# B&R Automation Studio project BR_ZBM1 (part 2)

#### Shiftregister.st - Shiftregister
```iecst
(********************************************************************
 * COPYRIGHT --
 ********************************************************************
 * Program: Shiftregister
 * File: ShiftregisterCyclic.st
 * Author: jorkes
 * Created: July 08, 2014
 ********************************************************************
 * Implementation of program Shiftregister
 ********************************************************************)

PROGRAM _INIT
	SHFTREG.typCounters.usChainCounter := 0;
	SHFTREG.typCounters.uiChainCnt16x16 := 0;
	SHFTREG.typCounters.usStartUpCntr := 0;
	SHFTREG.typCounters.bStartChainCntr := FALSE;
	bStartCnt := TRUE;

	//Preset
	SHFTREG.typCounters.usChainCounter := 0;
END_PROGRAM

PROGRAM _CYCLIC
	//==============================================================
	//Software met 2 x puls/grijper
	//Encoderpuls 1
	//==============================================================
	bEncPuls1 := FALSE;

	IF EDGENEG(MCU.typChain.status.bSetSpeedReached) THEN
		idxCntr := 0;
		bEncActive1 := FALSE;
	END_IF

	IF MCU.typChain.status.bSetSpeedReached OR TRUE THEN
		//#1
		IF EDGEPOS(MCU.typIN.bEncPuls1) AND NOT bEncActive1 THEN
			tiStop1 := T#0ms;
			tiStart1 := clock_ms();
			//Wacht weer op een volgende trigger. -> #2
			bEncActive1 := TRUE;

			//IF SHFTREG.typCounters.bStartChainCntr THEN
				//ringcounter 0-74
				//SHFTREG.typCounters.usChainCounter := (SHFTREG.typCounters.usChainCounter + 1) MOD (SHFTREG.uiGripperCnt);
			//END_IF

			//Meten van de gemiddelde tijd tussen twee grijpers.
//			IF NOT(bSubCounter) THEN
//				tiStart3 := tiStart1;
//				bSubCounter := TRUE;
//			ELSE
//				tiStop3 := tiStart1;
//				tiDiff3[idx_Diff3] := tiStop3 - tiStart3;
//
//				idx_Diff3 := (idx_Diff3 + 1) MOD 10;
//
//				tiDiff3Total := T#0ms;
//
//				FOR idx := 0 TO 9 DO
//					tiDiff3Total := tiDiff3Total + tiDiff3[idx];
//				END_FOR
//
//				tiDiff3Total := tiDiff3Total / 10;
//
//				IF idxCntr > 9 THEN
//					tiMusecSub := tiDiff3Total / 16;
//				ELSE
//					idxCntr := idxCntr + 1;
//					tiMusecSub := SHFTREG.tiDistanceBetweenGrippers / 16;
//				END_IF
//
//				bSubCounter := FALSE;
//			END_IF
		END_IF

		//Sla actuele tijd op.
		tiActual1 := clock_ms();

		//#2
		IF bEncActive1 THEN
			tiCheck1[idx_Diff1] := tiActual1 - tiStart1;
			//Controleer of de tweede puls van dezelfde grijper is en niet van de volgende.
			IF NOT(tiCheck1[idx_Diff1] > T#300ms) THEN
				//Als de volgende trigger binnen de 300ms valt dan is het dezelfde grijper.
				//IF EDGEPOS(MCU.typIN.bEncPuls1) THEN
				//	bStartEnc := TRUE;
				//END_IF
				//Controleer de trigger op de afgaande flank en sla de tijd op.
//				IF EDGENEG(MCU.typIN.bEncPuls1) THEN
//					tiStop1 := clock_ms();
//					tiDiff1 := tiStop1 - tiStart1;
//					//Als de tijd tussen opgaande en de afgaande flank groter is dan (100ms) genereer een puls met dubbele tijd.
//					IF tiDiff1 > T#100ms THEN
//						//Dubbele puls tijd.
//						//tpPulsEnc1.PT := T#10ms;
//						//Activeer puls.
//						//tpPulsEnc1.IN := TRUE;
//						//Wacht weer op een volgende trigger. -> #1
//						bEncActive1 := FALSE;
//						//Start de chaincounter bij de lange puls! -> #1
//						SHFTREG.typCounters.bStartChainCntr := TRUE;
//						//SHFTREG.typCounters.usChainCounter := 0;
//					END_IF
				IF EDGEPOS(MCU.typIN.bEncPuls1) THEN
					tiStop1 := clock_ms();
					tiDiff1 := tiStop1 - tiStart1;
					//Als de tijd tussen de twee triggerpulsen groter is dan (100ms) genereer een puls van 5ms.
					IF tiDiff1 > T#50ms THEN
						bEncPuls1 := TRUE;
						//Wacht weer op een volgende trigger. -> #1
						bEncActive1 := FALSE;
					END_IF
					idx_Diff1 := (idx_Diff1 + 1) MOD 75;
				ELSIF (tiCheck1[idx_Diff1] >= (T#149ms - T#30ms)) AND (tiStop1 = T#0ms) THEN //(T#149ms - T#30ms)) THEN
					// generate puls
					bEncPuls1 := TRUE;
					//Wacht weer op een volgende trigger. -> #1
					bEncActive1 := FALSE;
					//Start de chaincounter bij de lange puls! -> #1
					SHFTREG.typCounters.bStartChainCntr := TRUE;
					SHFTREG.typCounters.usChainCounter := 0;
					idx_Diff1 := (idx_Diff1 + 1) MOD 75;
				END_IF
			ELSE
				//Wacht weer op een volgende trigger. -> #1
				bEncActive1 := FALSE;
			END_IF
		END_IF
	END_IF

	IF EDGEPOS(bEncPuls1) THEN

		IF NOT(bSubCounter) THEN
			tiStart3 := clock_ms();
			bSubCounter := TRUE;
		ELSE
			tiStop3 := clock_ms();
			tiDiff3[idx_Diff3] := tiStop3 - tiStart3;

			idx_Diff3 := (idx_Diff3 + 1) MOD 10;

			tiDiff3Total := T#0ms;

			FOR idx := 0 TO 9 DO
				tiDiff3Total := tiDiff3Total + tiDiff3[idx];
			END_FOR

			tiDiff3Total := tiDiff3Total / 10;

			IF idxCntr > 9 THEN
				tiMusecSub := tiDiff3Total / 16;
			ELSE
				idxCntr := idxCntr + 1;
				tiMusecSub := SHFTREG.tiDistanceBetweenGrippers / 16;
			END_IF

			bSubCounter := FALSE;
		END_IF

		SHFTREG.typCounters.usChainCounter := (SHFTREG.typCounters.usChainCounter + 1) MOD (SHFTREG.uiGripperCnt);
	END_IF
		//#3
	IF EDGEPOS(MCU.typIN.bEncPuls2) AND NOT bEncActive2 THEN
		tiStart2 := clock_ms();
		//Wacht weer op een volgende trigger. -> #4
		bEncActive2 := TRUE;
	END_IF

	//Sla actuele tijd op.
	tiActual2 := clock_ms();

	//#4
	IF bEncActive2 THEN
		tiCheck2 := tiActual2 - tiStart2;
		//Controleer of de tweede puls van dezelfde grijper is en niet van de volgende.
		IF NOT(tiCheck2 > T#300ms) THEN
			//Als de volgende trigger binnen de 300ms valt dan is het dezelfde grijper.
			//Controleer de trigger op de afgaande flank en sla de tijd op.
			IF EDGENEG(MCU.typIN.bEncPuls2) THEN
				tiStop2 := clock_ms();
				tiDiff2 := tiStop2 - tiStart2;
				//Als de tijd tussen opgaande en de afgaande flank groter is dan (150ms) genereer een puls met dubbele tijd.
				IF tiDiff2 > T#100ms THEN
					//Dubbele puls tijd.
					tpPulsEnc2.PT := T#200ms;
					//Activeer puls.
					tpPulsEnc2.IN := TRUE;
					//Wacht weer op een volgende trigger. -> #3
					bEncActive2 := FALSE;
				END_IF
			ELSIF EDGEPOS(MCU.typIN.bEncPuls2) THEN
				tiStop2 := clock_ms();
				tiDiff2 := tiStop2 - tiStart2;
				//Als de tijd tussen de twee triggerpulsen groter is dan (50ms) genereer een puls van 100ms.
				IF tiDiff2 > T#50ms THEN
					//Dubbele puls tijd.
					tpPulsEnc2.PT := T#100ms;
					//Activeer puls.
					tpPulsEnc2.IN := TRUE;
					//Wacht weer op een volgende trigger. -> #3
					bEncActive2 := FALSE;
				END_IF
		END_IF		ELSE
			//Wacht weer op een volgende trigger. -> #3
			bEncActive2 := FALSE;
		END_IF
	END_IF

	PulsGenerator_0(tInit := bEncPuls1, enable := bGblSimulation OR MCU.typChain.status.bSetSpeedReached, sysTim := systemTime, tiHigh := T#1ms, tiLow := tiMusecSub);

	IF bEncPuls1 THEN
		SHFTREG.typCounters.uiChainCnt16x16 := SHFTREG.typCounters.uiChainCnt16x16 AND 240;
	END_IF

	IF EDGENEG(PulsGenerator_0.bOutput) THEN
		SHFTREG.typCounters.uiChainCnt16x16 := (SHFTREG.typCounters.uiChainCnt16x16 + 1) MOD 256;
		IF (SHFTREG.typCounters.uiChainCnt16x16 = 0) THEN
			SHFTREG.typCounters.usChainOffset := SHFTREG.typCounters.usChainCounter;
		END_IF
	END_IF

	//4 x cam & light triggers
	//	CamTrig_0(CamPos := 5, reset := MCU.typIN.bEncPuls1, trigger := EDGENEG(PulsGenerator_0.bOutput), tiPuls := T#30ms, tiDelay := T#15ms); //tiDelay = zie excel berekening Beschrijving software.xlsx
	//	CamTrig_1(CamPos := 10, reset := MCU.typIN.bEncPuls1, trigger := EDGENEG(PulsGenerator_0.bOutput), tiPuls := T#30ms, tiDelay := T#7ms);
	//	CamTrig_2(CamPos := 12, reset := MCU.typIN.bEncPuls1, trigger := EDGENEG(PulsGenerator_0.bOutput), tiPuls := T#30ms, tiDelay := T#11ms);
	//	CamTrig_3(CamPos := 2, reset := MCU.typIN.bEncPuls1, trigger := EDGENEG(PulsGenerator_0.bOutput), tiPuls := T#30ms, tiDelay := T#26ms);
	CamTrig_0(CamPos := Settings.CamPosition1, reset := bEncPuls1, trigger := EDGENEG(PulsGenerator_0.bOutput), tiPuls := INT_TO_TIME(Settings.CamPulseLength), tiDelay := INT_TO_TIME(Settings.CamDelay1), tiExtraLight := INT_TO_TIME(Settings.FlitsBefore)); //tiDelay = zie excel berekening Beschrijving software.xlsx
	CamTrig_1(CamPos := Settings.CamPosition2, reset := bEncPuls1, trigger := EDGENEG(PulsGenerator_0.bOutput), tiPuls := INT_TO_TIME(Settings.CamPulseLength), tiDelay := INT_TO_TIME(Settings.CamDelay2), tiExtraLight := INT_TO_TIME(Settings.FlitsBefore));
	CamTrig_2(CamPos := Settings.CamPosition3, reset := bEncPuls1, trigger := EDGENEG(PulsGenerator_0.bOutput), tiPuls := INT_TO_TIME(Settings.CamPulseLength), tiDelay := INT_TO_TIME(Settings.CamDelay3), tiExtraLight := INT_TO_TIME(Settings.FlitsBefore));
	CamTrig_3(CamPos := Settings.CamPosition4, reset := bEncPuls1, trigger := EDGENEG(PulsGenerator_0.bOutput), tiPuls := INT_TO_TIME(Settings.CamPulseLength), tiDelay := INT_TO_TIME(Settings.CamDelay4), tiExtraLight := INT_TO_TIME(Settings.FlitsBefore));

	MCU.typOUT.bLightTrigger1 := CamTrig_0.outLight;
	MCU.typOUT.bCamTrigger1 := CamTrig_0.outCam;
	MCU.typOUT.bLightTrigger2 := CamTrig_1.outLight;
	MCU.typOUT.bCamTrigger2 := CamTrig_1.outCam;
	MCU.typOUT.bLightTrigger3 := CamTrig_2.outLight;
	MCU.typOUT.bCamTrigger3 := CamTrig_2.outCam;
	MCU.typOUT.bLightTrigger4 := CamTrig_3.outLight;
	MCU.typOUT.bCamTrigger4 := CamTrig_3.outCam;

	//===============================
	//Software met kettingplaatjes
	//===============================
	//bEncPuls1 := MCU.typIN.bEncPuls1

	//Afhandelen van encodertrigger 1
//	IF EDGEPOS(bEncPuls1) AND NOT bFall_1 THEN
//		tiMusecStart4 := clock_ms();
//		IF toggle THEN
//			toggle := FALSE;
//			tiMusecStop3 := clock_ms();
//			tiMusecDiff3 := tiMusecStop3 - tiMusecStart1;
//			tiMusecSub := tiMusecDiff3 / 16;
//		END_IF
//
//		//get number of elapsed microseconds in current tick
//		tiMusecStart1 := clock_ms();
//
//		//Wait for first gripper (double length sensor puls)
//		IF SHFTREG.typCounters.bStartChainCntr THEN
//			//ringcounter 0-75
//			SHFTREG.typCounters.usChainCounter := (SHFTREG.typCounters.usChainCounter + 1) MOD (SHFTREG.uiGripperCnt);
//		ELSE
//			//startup counter. Only for completing average sensor measuring
//			SHFTREG.typCounters.usStartUpCntr := (SHFTREG.typCounters.usStartUpCntr + 1) MOD 255;
//		END_IF
//
//		//Variable prevends that falling edge is triggered first
//		bFall_1 := TRUE;
//	END_IF
//
//	IF EDGENEG(bEncPuls1) AND bFall_1 THEN
//		toggle := TRUE;
//
//		//get number of elapsed microseconds in current tick
//		tiMusecStop1 := clock_ms();
//		tiMusecDiff1 := tiMusecStop1 - tiMusecStart1;
//
//		AverageSens_0(index := SHFTREG.typCounters.usChainCounter, tiMeasure := tiMusecDiff1);
//
//		//First counter that takes care of detecting first gripper
//		IF SHFTREG.typCounters.usStartUpCntr > 9 THEN
//			AverageSens_0(enable := TRUE);
//			//Check if there was a 1.5 times of length of average sensor puls
//			//IF tiMusecDiff1 > ( (AverageSens_0.tiAverage * 3)/2) THEN
//			IF tiMusecDiff1 > ( (tiMusecDiff2 * 3)/2) THEN
//				tiMusecBetweenEncStart := clock_ms();
//				SHFTREG.typCounters.bStartChainCntr := TRUE;
//				SHFTREG.typCounters.usChainCounter := 0;
//			END_IF
//		END_IF
//
//		bFall_1 := FALSE;
//	END_IF
//
//	//Afhandelen van encodertrigger 2
//	IF EDGEPOS(bEncPuls2) AND NOT bFall_2 THEN
//		tiMusecStart2 := clock_ms();
//		bFall_2 := TRUE;
//	END_IF
//
//	IF EDGENEG(bEncPuls2) AND bFall_2 THEN
//		tiMusecStop2 := clock_ms();
//		tiMusecDiff2 := tiMusecStop2 - tiMusecStart2;
//
//		AverageSens_1(index := SHFTREG.typCounters.usChainCounter, tiMeasure := tiMusecDiff2);
//
//		//First counter that takes care of detecting first gripper
//		IF SHFTREG.typCounters.usStartUpCntr > 9 THEN
//			AverageSens_1(enable := TRUE);
//			//Check if there was a 1.5 times of length of average sensor puls
//			IF tiMusecDiff2 > ( (AverageSens_1.tiAverage * 3)/2) THEN
//				//Check if first sensor detected first gripper already
//
//				IF SHFTREG.typCounters.bStartChainCntr THEN
//					tiMusecBetweenEncStop := clock_ms();
//					//calculate time between encoder sensor, by measuring first grippper
//					tiMusecBetweenEncDiff[usCntr] := tiMusecBetweenEncStop - tiMusecBetweenEncStart;
//					usCntr := (usCntr + 1) MOD 100;
//				END_IF
//			END_IF
//		END_IF
//		bFall_2 := FALSE;
//	END_IF

	IF MCU.typInterface.State <> RUN THEN
		// Blink
		IF NOT tpBlink.Q THEN
			MCU.typOUT.bGreenLight := MCU.typOUT.bRedLight;
			MCU.typOUT.bRedLight := NOT MCU.typOUT.bRedLight;
		END_IF
		tpBlink(IN:=(NOT tpBlink.Q), PT:=T#500ms);
	ELSE
		IF bEncPuls1 THEN
			MCU.typOUT.bRedLight := TRUE;
			tiLastPuls := clock_ms();
		END_IF
		MCU.typOUT.bGreenLight := clock_ms() - tiLastPuls < T#400ms;
	END_IF

	// Reject Unit
	//usGripperIndex := ( SHFTREG.typCounters.usChainCounter + RU.usChainPos) MOD  SHFTREG.uiGripperCnt;
	usGripperIndex := ( SHFTREG.typCounters.usChainCounter + SHFTREG.uiGripperCnt - RU.usChainPos) MOD  SHFTREG.uiGripperCnt;
	IF SHFTREG.typGripper[usGripperIndex].bRejectActive THEN
		//RU.bAddFlower.SET1 := TRUE;
		IF RU.typSettings.usTimingBU16 MOD 16 = SHFTREG.typCounters.uiChainCnt16x16 MOD 16 THEN
			RU.typOUT.bActivateGripper := SHFTREG.typGripper[usGripperIndex].bRejectOnOff;
			//fbResetGripper( ThisGripper := SHFTREG.typGripper[usGripperIndex]);
			SHFTREG.typGripper[usGripperIndex].bRejectActive := FALSE;
			SHFTREG.typGripper[usGripperIndex].bRejectOnOff := FALSE;
		END_IF
	END_IF

	// Now check if a gripper is positioned for the BU
	FOR i := 0 TO 9 DO

		//JORKES
		usGripperIndex := ( SHFTREG.typCounters.usChainCounter + SHFTREG.uiGripperCnt - BU[i].usChainPos) MOD  SHFTREG.uiGripperCnt;

		IF NOT BU[i].typInterface.bEmptyCmd THEN
			BU[i].typInterface.bEmptyCmd := SHFTREG.typGripper[usGripperIndex].siEmptyBU = i;
			SHFTREG.typGripper[usGripperIndex].siEmptyBU := -1;
			AsArLogWrite_EmptyCmd(enable := TRUE, ident := arlogBASE_USER_LOG_IDENT, logLevel := 1, errornr := 50003, mem := ADR(i), len := SIZEOF(i), asciiString :=  ADR('Empty command received'));
		END_IF

		IF NOT BU[i].bAddFlower THEN
			//JORKES
			//usGripperIndex := ( SHFTREG.typCounters.usChainCounter + SHFTREG.uiGripperCnt - BU[i].usChainPos) MOD  SHFTREG.uiGripperCnt;
			BU[i].GripperControl.IN := FALSE;

			//IF EDGEPOS(BU[i].typInterface.bEmptyCmd) THEN
			//	AsArLogWrite_EmptyCmd(enable := TRUE, ident := arlogBASE_USER_LOG_IDENT, logLevel := 1, errornr := 50002, mem := 0, len := 0, asciiString :=  ADR('Bosunit empty cmd set'));
			//END_IF

			IF i = SHFTREG.typGripper[usGripperIndex].usSetTarget THEN
				//SHFTREG.typGripper[usGripperIndex].
				BU[i].bAddFlower := TRUE;
				BU[i].typInterface.iReceivePos := SHFTREG.typGripper[usGripperIndex].uiCorrection;
				IF SHFTREG.typGripper[usGripperIndex].bFast THEN
					BU[i].typInterface.usServoSpeed := BU[i].typSettings.usFastSpeed;
				ELSE
					BU[i].typInterface.usServoSpeed := BU[i].typSettings.usSpeed;
				END_IF
				//////////BU[i].typSettings.usTimingBU16 := INT_TO_SINT( SHFTREG.typGripper[usGripperIndex].uiTimingBU16 MOD 16);
				// The gripper data is assigend
				//IF EDGEPOS(BU[i].bAddFlower) THEN
				//	AsArLogWrite_EmptyCmd(enable := TRUE, ident := arlogBASE_USER_LOG_IDENT, logLevel := 1, errornr := 50003, mem := ADR(i), len := SIZEOF(i), asciiString :=  ADR('Add flower'));
				//END_IF
			ELSE
				// The first gripper doen's contain a flow, does the
				usGripperIndex := ( SHFTREG.typCounters.usChainCounter - 1 + BU[i].usChainPos) MOD SHFTREG.uiGripperCnt;
				IF i = SHFTREG.typGripper[usGripperIndex].usSetTarget AND NOT BU[i].bBusyDrop THEN
					BU[i].typInterface.iReceivePos := SHFTREG.typGripper[usGripperIndex].uiCorrection;
				END_IF
			END_IF
		ELSE IF NOT BU[i].bBusyDrop THEN
			//JORKES
			//IF EDGEPOS(BU[i].rsActivateGripper.Q1) THEN
			IF EDGEPOS(BU[i].typSettings.usTimingBU16 = (SHFTREG.typCounters.uiChainCnt16x16 MOD 16) ) AND (i = SHFTREG.typGripper[usGripperIndex].usSetTarget) THEN
				fbResetGripper( ThisGripper := SHFTREG.typGripper[usGripperIndex]);
				BU[i].GripperControl.IN := TRUE;
				BU[i].bAddFlower := FALSE;
				END_IF
			END_IF

			//JORKES
			//BU[i].GripperControl.IN :=  BU[i].rsActivateGripper.Q1; // AND  i = SHFTREG.typGripper[usGripperIndex].usSetTarget;
			//BU[i].GripperControl.IN :=  BU[i].typSettings.usTimingBU16 = SHFTREG.typCounters.uiChainCnt16x16 MOD 16; // AND  i = SHFTREG.typGripper[usGripperIndex].usSetTarget;
		END_IF

		IF EDGENEG(BU[i].typOUT.bActivateGripper) THEN
		//	BU[i].bAddFlower(SET1 := FALSE, RESET := TRUE);
		END_IF
		//BU[i].GripperControl(tiSensDelay := BU[i].typInterface.tiDelayActiveGripper, tiSensPuls := INT_TO_TIME( Settings.BU_ActivateReleaseTime )); // T#3000ms); // Was 100 RSP
		BU[i].GripperControl( PT := INT_TO_TIME( Settings.BU_ActivateReleaseTime ));
		BU[i].typOUT.bActivateGripper := BU[i].GripperControl.Q OR  BU[i].typInterface.bManualGripperCmd;
		//JORKES
		//BU[i].rsActivateGripper(RESET1 := NOT BU[i].bAddFlower);
		//BU[i].GripperControl.IN :=  BU[i].rsActivateGripper.Q1;

		// TO DO
		// BU[i].bAddFlower.RESET := (i = SHFTREG.typGripper[usGripperIndex].usSetTarget);

	END_FOR
END_PROGRAM
```

#### Shiftregister.var - Local variables
```iecst
(********************************************************************
 * COPYRIGHT --
 ********************************************************************
 * Program: Shiftregister
 * File: Shiftregister.var
 * Author: jorkes
 * Created: July 08, 2014
 ********************************************************************
 * Local variables of program Shiftregister
 ********************************************************************)
(*Log*)
VAR
	AsArLogWrite_EmptyCmd : AsArLogWrite := (0);
	tiLastPuls : TIME;
END_VAR
(*Zonder kettingplaatjes*)
VAR
	bSubCounter : BOOL := FALSE;
	bEncPuls2 : BOOL;
	bEncPuls1 : BOOL;
	tpPulsEnc2 : TP;
	tpPulsEnc1 : TP;
	bEncActive1 : BOOL;
	bEncActive2 : BOOL;
	idxCntr : USINT := 0;
	idx : USINT := 0;
	idx_Diff1 : USINT := 0;
	idx_Diff3 : USINT := 0;
	tiActual2 : TIME;
	tiActual1 : TIME;
	tiCheck1 : ARRAY[0..74] OF TIME;
	tiDiff1 : TIME;
	tiStop1 : TIME;
	tiStart1 : TIME;
	tiCheck2 : TIME;
	tiDiff2 : TIME;
	tiStop2 : TIME;
	tiStart2 : TIME;
	tiCheck3 : TIME;
	tiDiff3Total : TIME;
	tiDiff3 : ARRAY[0..9] OF TIME;
	tiStop3 : TIME;
	tiStart3 : TIME;
END_VAR
(*Kettingteller*)
VAR
	bFall_1 : BOOL := FALSE;
	bFall_2 : BOOL := FALSE;
	tiMusecDiff2 : TIME;
	tiMusecDiff1 : TIME;
	tiMusecStart2 : TIME;
	tiMusecStart1 : TIME;
	tiMusecStop2 : TIME;
	tiMusecStop1 : TIME;
END_VAR
(*Kettingrek*)
VAR
	usCntr : USINT := 0;
	tiMusecBetweenEncDiff : ARRAY[0..100] OF TIME;
	tiMusecBetweenEncStop : TIME;
	tiMusecBetweenEncStart : TIME;
	AverageSens_1 : fbAverage;
	AverageSens_0 : fbAverage;
END_VAR
(*Grijper*)
VAR
	tiMusecSub : TIME := T#600ms;
	tiMusecDiff3 : TIME;
	tiMusecStop3 : TIME;
	toggle : BOOL;
END_VAR
(*Subcounter*)
VAR
	bStartCnt : BOOL;
	tiMusecDiff4 : TIME;
	tiMusecActual4 : TIME;
	PulsGenerator_0 : PulsGenerator;
	tiMusecStart4 : TIME;
	CamTrig_0 : fbTriggerBuf;
	CamTrig_1 : fbTriggerBuf;
	CamTrig_2 : fbTriggerBuf;
	CamTrig_3 : fbTriggerBuf;
END_VAR
(*Ligths*)
VAR
	tpBlink : TP;
END_VAR
(*BunchUnits*)
VAR
	i : USINT;
	usGripperIndex : USINT;
END_VAR
```

#### Shiftregister1.st - not listed in the package file held
```iecst
(********************************************************************
 * COPYRIGHT --
 ********************************************************************
 * Program: Shiftregister
 * File: ShiftregisterCyclic.st
 * Author: jorkes
 * Created: July 08, 2014
 ********************************************************************
 * Implementation of program Shiftregister
 ********************************************************************)

PROGRAM _INIT
	SHFTREG.typCounters.usChainCounter := 0;
	SHFTREG.typCounters.uiChainCnt16x16 := 0;
	SHFTREG.typCounters.usStartUpCntr := 0;
	SHFTREG.typCounters.bStartChainCntr := FALSE;
	bStartCnt := TRUE;
END_PROGRAM

PROGRAM _CYCLIC
	PulsGenerator_0(tInit := MCU.typIN.bEncPuls1, enable := bGblSimulation OR MCU.typInterface.State = RUN, sysTim := systemTime, tiHigh := T#1ms, tiLow := tiMusecSub);

	IF EDGENEG(PulsGenerator_0.bOutput) THEN
		SHFTREG.typCounters.uiChainCnt16x16 := (SHFTREG.typCounters.uiChainCnt16x16 + 1) MOD 256;
		IF (SHFTREG.typCounters.uiChainCnt16x16 = 0) THEN
			SHFTREG.typCounters.usChainOffset := SHFTREG.typCounters.usChainCounter;
		END_IF
	END_IF

	//4 x cam & light triggers
//	CamTrig_0(CamPos := 5, reset := MCU.typIN.bEncPuls1, trigger := EDGENEG(PulsGenerator_0.bOutput), tiPuls := T#30ms, tiDelay := T#15ms); //tiDelay = zie excel berekening Beschrijving software.xlsx
//	CamTrig_1(CamPos := 10, reset := MCU.typIN.bEncPuls1, trigger := EDGENEG(PulsGenerator_0.bOutput), tiPuls := T#30ms, tiDelay := T#7ms);
//	CamTrig_2(CamPos := 12, reset := MCU.typIN.bEncPuls1, trigger := EDGENEG(PulsGenerator_0.bOutput), tiPuls := T#30ms, tiDelay := T#11ms);
//	CamTrig_3(CamPos := 2, reset := MCU.typIN.bEncPuls1, trigger := EDGENEG(PulsGenerator_0.bOutput), tiPuls := T#30ms, tiDelay := T#26ms);
	CamTrig_0(CamPos := Settings.CamPosition1, reset := MCU.typIN.bEncPuls1, trigger := EDGENEG(PulsGenerator_0.bOutput), tiPuls := INT_TO_TIME(Settings.CamPulseLength), tiDelay := INT_TO_TIME(Settings.CamDelay1), tiExtraLight := INT_TO_TIME(Settings.FlitsBefore)); //tiDelay = zie excel berekening Beschrijving software.xlsx
	CamTrig_1(CamPos := Settings.CamPosition2, reset := MCU.typIN.bEncPuls1, trigger := EDGENEG(PulsGenerator_0.bOutput), tiPuls := INT_TO_TIME(Settings.CamPulseLength), tiDelay := INT_TO_TIME(Settings.CamDelay2), tiExtraLight := INT_TO_TIME(Settings.FlitsBefore));
	CamTrig_2(CamPos := Settings.CamPosition3, reset := MCU.typIN.bEncPuls1, trigger := EDGENEG(PulsGenerator_0.bOutput), tiPuls := INT_TO_TIME(Settings.CamPulseLength), tiDelay := INT_TO_TIME(Settings.CamDelay3), tiExtraLight := INT_TO_TIME(Settings.FlitsBefore));
	CamTrig_3(CamPos := Settings.CamPosition4, reset := MCU.typIN.bEncPuls1, trigger := EDGENEG(PulsGenerator_0.bOutput), tiPuls := INT_TO_TIME(Settings.CamPulseLength), tiDelay := INT_TO_TIME(Settings.CamDelay4), tiExtraLight := INT_TO_TIME(Settings.FlitsBefore));

	MCU.typOUT.bLightTrigger1 := CamTrig_0.outLight;
	MCU.typOUT.bCamTrigger1 := CamTrig_0.outCam;
	MCU.typOUT.bLightTrigger2 := CamTrig_1.outLight;
	MCU.typOUT.bCamTrigger2 := CamTrig_1.outCam;
	MCU.typOUT.bLightTrigger3 := CamTrig_2.outLight;
	MCU.typOUT.bCamTrigger3 := CamTrig_2.outCam;
	MCU.typOUT.bLightTrigger4 := CamTrig_3.outLight;
	MCU.typOUT.bCamTrigger4 := CamTrig_3.outCam;

	//Afhandelen van encodertrigger 1
	IF EDGEPOS(MCU.typIN.bEncPuls1) AND NOT bFall_1 THEN
		tiMusecStart4 := clock_ms();
		IF toggle THEN
			toggle := FALSE;
			tiMusecStop3 := clock_ms();
			tiMusecDiff3 := tiMusecStop3 - tiMusecStart1;
			tiMusecSub := tiMusecDiff3 / 16;
		END_IF

		//get number of elapsed microseconds in current tick
		tiMusecStart1 := clock_ms();

		//Wait for first gripper (double length sensor puls)
		IF SHFTREG.typCounters.bStartChainCntr THEN
			//ringcounter 0-75
			SHFTREG.typCounters.usChainCounter := (SHFTREG.typCounters.usChainCounter + 1) MOD (SHFTREG.uiGripperCnt);
		ELSE
			//startup counter. Only for completing average sensor measuring
			SHFTREG.typCounters.usStartUpCntr := (SHFTREG.typCounters.usStartUpCntr + 1) MOD 255;
		END_IF

		//Variable prevends that falling edge is triggered first
		bFall_1 := TRUE;
	END_IF

	IF EDGENEG(MCU.typIN.bEncPuls1) AND bFall_1 THEN
		toggle := TRUE;

		//get number of elapsed microseconds in current tick
		tiMusecStop1 := clock_ms();
		tiMusecDiff1 := tiMusecStop1 - tiMusecStart1;

		AverageSens_0(index := SHFTREG.typCounters.usChainCounter, tiMeasure := tiMusecDiff1);

		//First counter that takes care of detecting first gripper
		IF SHFTREG.typCounters.usStartUpCntr > 9 THEN
			AverageSens_0(enable := TRUE);
			//Check if there was a 1.5 times of length of average sensor puls
			IF tiMusecDiff1 > ( (AverageSens_0.tiAverage * 3)/2) THEN
				tiMusecBetweenEncStart := clock_ms();
				SHFTREG.typCounters.bStartChainCntr := TRUE;
			END_IF
		END_IF

		bFall_1 := FALSE;
	END_IF

	//Afhandelen van encodertrigger 2
	IF EDGEPOS(MCU.typIN.bEncPuls2) AND NOT bFall_2 THEN
		tiMusecStart2 := clock_ms();
		bFall_2 := TRUE;
	END_IF

	IF EDGENEG(MCU.typIN.bEncPuls2) AND bFall_2 THEN
		tiMusecStop2 := clock_ms();
		tiMusecDiff2 := tiMusecStop2 - tiMusecStart2;

		AverageSens_1(index := SHFTREG.typCounters.usChainCounter, tiMeasure := tiMusecDiff2);

		//First counter that takes care of detecting first gripper
		IF SHFTREG.typCounters.usStartUpCntr > 9 THEN
			AverageSens_1(enable := TRUE);
			//Check if there was a 1.5 times of length of average sensor puls
			IF tiMusecDiff2 > ( (AverageSens_1.tiAverage * 3)/2) THEN
				//Check if first sensor detected first gripper already
				IF SHFTREG.typCounters.bStartChainCntr THEN
					tiMusecBetweenEncStop := clock_ms();
					//calculate time between encoder sensor, by measuring first grippper
					tiMusecBetweenEncDiff[usCntr] := tiMusecBetweenEncStop - tiMusecBetweenEncStart;
					usCntr := (usCntr + 1) MOD 100;
				END_IF
			END_IF
		END_IF
		bFall_2 := FALSE;
	END_IF

	IF MCU.typInterface.State <> RUN THEN
		// Blink
		IF NOT tpBlink.Q THEN
			MCU.typOUT.bGreenLight := MCU.typOUT.bRedLight;
			MCU.typOUT.bRedLight := NOT MCU.typOUT.bRedLight;
		END_IF
		tpBlink(IN:=(NOT tpBlink.Q), PT:=T#500ms);
	ELSE
		MCU.typOUT.bRedLight := (MCU.typIN.bEncPuls1);
		MCU.typOUT.bGreenLight := TRUE;
	END_IF

	// Reject Unit
	//usGripperIndex := ( SHFTREG.typCounters.usChainCounter + RU.usChainPos) MOD  SHFTREG.uiGripperCnt;
	usGripperIndex := ( SHFTREG.typCounters.usChainCounter + SHFTREG.uiGripperCnt - RU.usChainPos) MOD  SHFTREG.uiGripperCnt;
	IF SHFTREG.typGripper[usGripperIndex].bRejectActive THEN
		//RU.srAddFlower.SET1 := TRUE;
		IF RU.typSettings.usTimingBU16 MOD 16 = SHFTREG.typCounters.uiChainCnt16x16 MOD 16 THEN
			RU.typOUT.bActivateGripper := SHFTREG.typGripper[usGripperIndex].bRejectOnOff;
			//fbResetGripper( ThisGripper := SHFTREG.typGripper[usGripperIndex]);
			SHFTREG.typGripper[usGripperIndex].bRejectActive := FALSE;
			SHFTREG.typGripper[usGripperIndex].bRejectOnOff := FALSE;
		END_IF
	END_IF

	// Now check if a gripper is positioned for the BU
	FOR i := 0 TO 1 DO

		usGripperIndex := ( SHFTREG.typCounters.usChainCounter + SHFTREG.uiGripperCnt - BU[i].usChainPos) MOD  SHFTREG.uiGripperCnt;
		//IF BU[i].typSettings.usTimingBU16 = SHFTREG.typCounters.uiChainCnt16x16 MOD 16 AND  i = SHFTREG.typGripper[usGripperIndex].usSetTarget THEN
		// The time has come to activate the grippers!!!
		//	BU[i].GripperControl.IN := TRUE;
		//END_IF

		IF NOT BU[i].srAddFlower THEN
			usGripperIndex := ( SHFTREG.typCounters.usChainCounter + SHFTREG.uiGripperCnt - BU[i].usChainPos) MOD  SHFTREG.uiGripperCnt;
		//	IF i = SHFTREG.typGripper[usGripperIndex].usSetTarget THEN
		//		// The first gripper doen's contain a flow, does the
		//		usGripperIndex := ( SHFTREG.typCounters.usChainCounter - 1 + BU[i].usChainPos) MOD  SHFTREG.uiGripperCnt;
		//		BU[i].typInterface.iReceivePos := SHFTREG.typGripper[usGripperIndex].uiCorrection;
		//	END_IF

			IF i = SHFTREG.typGripper[usGripperIndex].usSetTarget THEN
				//SHFTREG.typGripper[usGripperIndex].
				BU[i].srAddFlower := TRUE;
				BU[i].typInterface.bEmptyCmd := SHFTREG.typGripper[usGripperIndex].bEmptyBU;
				BU[i].typInterface.iReceivePos := SHFTREG.typGripper[usGripperIndex].uiCorrection;
				IF SHFTREG.typGripper[usGripperIndex].bFast THEN
					BU[i].typInterface.usServoSpeed := BU[i].typSettings.usFastSpeed;
				ELSE
					BU[i].typInterface.usServoSpeed := BU[i].typSettings.usSpeed;
				END_IF
				//////////BU[i].typSettings.usTimingBU16 := INT_TO_SINT( SHFTREG.typGripper[usGripperIndex].uiTimingBU16 MOD 16);
				// The gripper data is assigend

			END_IF
		ELSE
			// BU[i].srAddFlower.Q1 = TRUE so a flower is already assigned
			usGripperIndex := ( SHFTREG.typCounters.usChainCounter + SHFTREG.uiGripperCnt - BU[i].usChainPos) MOD  SHFTREG.uiGripperCnt;
			BU[i].rsActivateGripper.SET := BU[i].typSettings.usTimingBU16 = SHFTREG.typCounters.uiChainCnt16x16 MOD 16  AND  i = SHFTREG.typGripper[usGripperIndex].usSetTarget;

			//IF BU[i].typSettings.usTimingBU16 = SHFTREG.typCounters.uiChainCnt16x16 MOD 16 AND  i = SHFTREG.typGripper[usGripperIndex].usSetTarget THEN
				// The time has come to activate the grippers!!!
			//	BU[i].GripperControl.IN := TRUE;
			//END_IF
			IF EDGEPOS(BU[i].rsActivateGripper.Q1) THEN
				fbResetGripper( ThisGripper := SHFTREG.typGripper[usGripperIndex]);
			END_IF
			BU[i].GripperControl.IN :=  BU[i].rsActivateGripper.Q1; // AND  i = SHFTREG.typGripper[usGripperIndex].usSetTarget;
			//BU[i].GripperControl.IN :=  BU[i].typSettings.usTimingBU16 = SHFTREG.typCounters.uiChainCnt16x16 MOD 16; // AND  i = SHFTREG.typGripper[usGripperIndex].usSetTarget;
		END_IF

		IF EDGENEG(BU[i].typOUT.bActivateGripper) THEN
		//	BU[i].srAddFlower(SET1 := FALSE, RESET := TRUE);
		END_IF
		//BU[i].GripperControl(tiSensDelay := BU[i].typInterface.tiDelayActiveGripper, tiSensPuls := INT_TO_TIME( Settings.BU_ActivateReleaseTime )); // T#3000ms); // Was 100 RSP
		BU[i].GripperControl( PT := INT_TO_TIME( Settings.BU_ActivateReleaseTime ));
		BU[i].typOUT.bActivateGripper := BU[i].GripperControl.Q;
		BU[i].rsActivateGripper(RESET1 := NOT BU[i].srAddFlower);
		BU[i].GripperControl.IN :=  BU[i].rsActivateGripper.Q1;;
		// TO DO
		// 							BU[i].srAddFlower.RESET := (i = SHFTREG.typGripper[usGripperIndex].usSetTarget);

	END_FOR
END_PROGRAM
```

### Program Logical/MainControlUnit/Simulation (IEC) - Program

#### Simulation.st - Implementation code
```iecst
(********************************************************************
 * COPYRIGHT --
 ********************************************************************
 * Program: Simulation
 * File: Simulation.st
 * Author: jorkes
 * Created: July 08, 2014
 ********************************************************************
 * Implementation of program Init
 ********************************************************************)

PROGRAM _INIT
	typEncPuls1.tiHigh := tiEncPulsShort;
	typEncPuls1.tiLow := SHFTREG.tiDistanceBetweenGrippers - tiEncPulsShort;

	typEncPuls2.tiHigh := tiEncPulsShort;
	typEncPuls2.tiLow := SHFTREG.tiDistanceBetweenGrippers - tiEncPulsShort;
END_PROGRAM

PROGRAM _CYCLIC
	typEncPuls1(enable := bGblSimulation, sysTim := systemTime);
	typEncPuls2(enable := bGblSimulation, sysTim := systemTime);

	// In simulation the pulses are generated by the above function.
	IF bGblSimulation THEN
		MCU.typIN.bEncPuls1 := typEncPuls1.bOutput;
		MCU.typIN.bEncPuls2 := typEncPuls2.bOutput;
	END_IF

	IF SHFTREG.typCounters.bStartChainCntr THEN
		IF  SHFTREG.typCounters.usChainCounter >= (SHFTREG.uiGripperCnt - 1) THEN
			typEncPuls1.tiHigh := tiEncPulsLong;
			typEncPuls1.tiLow := SHFTREG.tiDistanceBetweenGrippers - tiEncPulsLong;
		ELSE
			typEncPuls1.tiHigh := tiEncPulsShort;
			typEncPuls1.tiLow := SHFTREG.tiDistanceBetweenGrippers - tiEncPulsShort;
		END_IF
	ELSE
		IF  SHFTREG.typCounters.usStartUpCntr >= 10 THEN
			typEncPuls1.tiHigh := tiEncPulsLong;
			typEncPuls1.tiLow := SHFTREG.tiDistanceBetweenGrippers - tiEncPulsLong;
		ELSE
			typEncPuls1.tiHigh := tiEncPulsShort;
			typEncPuls1.tiLow := SHFTREG.tiDistanceBetweenGrippers - tiEncPulsShort;
		END_IF
	END_IF

	IF SHFTREG.typCounters.usChainCounter = SHFTREG.typEncoder.uiEncSensorPosition2 THEN //Aantal grijpers tussen eerste en tweede encoder.
		typEncPuls2.tiHigh := tiEncPulsLong;
		typEncPuls2.tiLow := SHFTREG.tiDistanceBetweenGrippers - tiEncPulsLong;
	ELSE
		typEncPuls2.tiHigh := tiEncPulsShort;
		typEncPuls2.tiLow := SHFTREG.tiDistanceBetweenGrippers - tiEncPulsShort;
	END_IF

	//4 x cam & light triggers
	//Sensor_0(trigger := MCU.typIN.bEncPuls1, tiPuls := tiPulsCam, tiDelay := tiDelayCam_0);
	//Sensor_1(trigger := MCU.typIN.bEncPuls1, tiPuls := tiPulsCam, tiDelay := tiDelayCam_1);
	//Sensor_2(trigger := MCU.typIN.bEncPuls1, tiPuls := tiPulsCam, tiDelay := tiDelayCam_2);
	//Sensor_3(trigger := MCU.typIN.bEncPuls1, tiPuls := tiPulsCam, tiDelay := tiDelayCam_3);

	//MCU.typOUT.bCamTrigger1 := Sensor_0.outCam;
	//MCU.typOUT.bCamTrigger2 := Sensor_1.outCam;
	//MCU.typOUT.bCamTrigger3 := Sensor_2.outCam;
	//MCU.typOUT.bCamTrigger4 := Sensor_3.outCam;

	//MCU.typOUT.bLightTrigger1 := Sensor_0.outLight;
	//MCU.typOUT.bLightTrigger2 := Sensor_1.outLight;
	//MCU.typOUT.bLightTrigger3 := Sensor_2.outLight;
	//MCU.typOUT.bLightTrigger4 := Sensor_3.outLight;
END_PROGRAM
```

#### Simulation.var - Local variables
```iecst
(********************************************************************
 * COPYRIGHT --
 ********************************************************************
 * Program: Init
 * File: Init.var
 * Author: jorkes
 * Created: July 08, 2014
 ********************************************************************
 * Local variables of program Init
 ********************************************************************)
VAR
	typEncPuls2 : PulsGenerator;
	typEncPuls1 : PulsGenerator;
	tiEncPulsLong : TIME := T#100ms;
	tiEncPulsShort : TIME := T#50ms;
END_VAR
(*Camtriggers*)
VAR
	tiDelayCam_0 : TIME := T#200ms;
	tiDelayCam_1 : TIME := T#400ms;
	tiDelayCam_2 : TIME := T#450ms;
	tiDelayCam_3 : TIME := T#100ms;
	tiPulsCam : TIME := T#20ms;
	Sensor_0 : fbTriggerBuf;
	Sensor_1 : fbTriggerBuf;
	Sensor_2 : fbTriggerBuf;
	Sensor_3 : fbTriggerBuf;
END_VAR
```

### Program Logical/MainControlUnit/Main (IEC) - Program

#### Main.st - Implementation code
```iecst
(********************************************************************
 * COPYRIGHT --
 ********************************************************************
 * Program: Main
 * File: Main.st
 * Author: jorkes
 * Created: August 14, 2014
 ********************************************************************
 * Implementation of program Main
 ********************************************************************)

PROGRAM _CYCLIC
	//TestPuls(tiHigh := T#40ms, tiLow := T#20ms);
	MCU.motChain.bResetFault := FALSE;
	MBU.motKnifeUnit.bResetFault := FALSE;
	MCU.typOUT.bBuzzer := FALSE;

	// If software toggle is activated, override the input.
	IF MCU.typInterface.bToggle THEN
		MCU.typIN.bJog := MCU.typInterface.bToggle;
	END_IF

	IF EDGEPOS(MCU.typIN.bJog) THEN
		MCU.motChain.iSpeed := MCU.typInterface.iJogSpeed;
		MCU.motChain.bResetFault := TRUE;
	END_IF

	IF EDGENEG(MCU.typIN.bJog) OR EDGEPOS(MCU.typInterface.bRun) THEN
		MCU.motChain.iSpeed := MCU.typInterface.iNormalSpeed;
		MCU.motChain.bResetFault := TRUE;
		MBU.motKnifeUnit.bResetFault := TRUE;
	END_IF

	IF EDGENEG(MCU.typInterface.bRun) THEN

		iBUEnabledMask := -1;
		FOR i := 0 TO 9 BY 1 DO
			//
			BU[i].typInterface.bEnable := FALSE;
		END_FOR

		IF  MCU.typChain.status.bFault THEN
			// Reset drive
			MCU.motChain.bResetFault := TRUE;
		END_IF
	END_IF

	IF MCU.typInterface.bReset THEN
		MCU.motChain.bResetFault := TRUE;
		MBU.motKnifeUnit.bResetFault := TRUE;
		MCU.typInterface.bReset := FALSE;
		MCU.typInterface.bRun := FALSE;
	ELSE
		IF  MCU.typInterface.bRun  THEN
			//
			IF MCU.typInterface.iBUEnabledMask <> iBUEnabledMask THEN
				iBUEnabledMask := MCU.typInterface.iBUEnabledMask;
				FOR i := 0 TO 9 BY 1 DO
					//
					iOut := SHL(iMask, i);
					BU[i].typInterface.bEnable :=  (iMask AND iBUEnabledMask) = 0;
					//BU[i].typInterface.bEnable :=  (SHL(1, i) AND iBUEnabledMask) = 0;
				END_FOR

			END_IF
			IF MCU.typInterface.bEmpty THEN
				// Start empty machine
				IF MCU.typInterface.bIsEmpty THEN
					MCU.typInterface.bRun := FALSE;
				END_IF
			ELSE
				// Normal RUN
				IF MCU.typChain.status.bRun THEN
					MCU.typInterface.State := RUN;
				ELSE
					IF MCU.typChain.status.bFault THEN
						// Drive in error remove command
						MCU.typInterface.bRun := FALSE;
					ELSE
						bRunRequest := TRUE;
					END_IF
				END_IF
			END_IF
		ELSE
			// bRun is False.
			bRunRequest := FALSE;
			MCU.typInterface.bEmpty := FALSE;
		END_IF
	END_IF

	CASE MCU.typInterface.State OF
		RUN: // Start main motor
			IF MCU.typChain.status.bFault = TRUE OR NOT MCU.typInterface.bRun THEN
				MCU.typInterface.State := STOP;
			ELSE
				MCU.typChain.command.bPower := TRUE;
				bRunRequest := TRUE;
				IF MCU.typChain.status.bSetSpeedReached THEN
					MCU.typInterface.State := RUN;
				END_IF
			END_IF
		STOP:
			bRunRequest := FALSE;
			bGblSimulation := FALSE;
			IF 	MCU.typInterface.bRun THEN
				IF NOT MCU.typInterface.bSimulation THEN
					MCU.typInterface.State := RUN;
				ELSE
					MCU.typInterface.State := SIMULATION;
				END_IF
			END_IF
		EMPTY:
			IF MCU.typChain.status.bFault = TRUE THEN
				MCU.typInterface.State := STOP;
			ELSE
				MCU.typInterface.State := EMPTY;
			END_IF

		SIMULATION:
			bGblSimulation := MCU.typInterface.bEnabled AND  MCU.typInterface.bSimulation;
			IF NOT MCU.typInterface.bRun THEN
				MCU.typInterface.State := STOP;
				bGblSimulation := FALSE;
			ELSE
				MCU.typInterface.State := SIMULATION;
			END_IF
	END_CASE
	// END_IF

	//tonStart(IN := MCU.typInterface.bRun, PT := T#3s);
	// When starting the chain, first sound a zoomer.
	tonStart(IN := bRunRequest OR MCU.typIN.bJog, PT := T#3s);
	tonJogDelay(IN := (srJogDelay.Q1 AND NOT  MCU.typIN.bJog) , PT := T#5s);
	srJogDelay( SET1 := EDGENEG( MCU.typIN.bJog), RESET := tonJogDelay.Q AND NOT (bRunRequest OR MCU.typIN.bJog));
	bRunRequest := tonStart.Q;
	IF  (srJogDelay.Q1) AND NOT bRunRequest THEN
		bRunRequest := bRunRequest OR MCU.typIN.bJog;
	END_IF

	MCU.typOUT.bBuzzer := bRunRequest <> tonStart.IN OR MCU.typInterface.bBuzzer;
	// If the MCU.typInterface.bBuzzer is not reset in 5 sec. The auto reset zoomer.
	tonBuzzerReset( IN := MCU.typInterface.bBuzzer, PT := T#5s);
	IF( tonBuzzerReset.Q ) THEN
		MCU.typInterface.bBuzzer := FALSE;
	END_IF

	// Set the command to the drive
	MCU.motChain.bRun := bRunRequest;
	MCU.motChain.bRunReverse := FALSE;
	MCU.motChain( MotorStruc := MCU.typChain);

	//JORKES 18022015
	//Camera trigger manual
	IF MCU.typInterface.State = STOP THEN
		//Use bBuzzer for triggering camera's when machine is in STOP or PAUZE state.
		//MCU.typInterface.bCamTrigManual := MCU.typInterface.bBuzzer;

		//Create light triggers.
		tpLightTrig1(IN := MCU.typInterface.bCamTrigManual, PT := tiLightPuls);
		tpLightTrig2(IN := EDGENEG(tpLightTrig1.Q), PT := tiLightPuls);
		tpLightTrig3(IN := EDGENEG(tpLightTrig2.Q), PT := tiLightPuls);
		tpLightTrig4(IN := EDGENEG(tpLightTrig3.Q), PT := tiLightPuls);

		//Create cam triggers.
		tpCamTrig1(IN := EDGEPOS(tpLightTrig1.ET >= T#10ms), PT := tiCamPuls);
		tpCamTrig2(IN := EDGEPOS(tpLightTrig2.ET >= T#10ms), PT := tiCamPuls);
		tpCamTrig3(IN := EDGEPOS(tpLightTrig3.ET >= T#10ms), PT := tiCamPuls);
		tpCamTrig4(IN := EDGEPOS(tpLightTrig4.ET >= T#10ms), PT := tiCamPuls);

		//Set outputs for light's.
		MCU.typOUT.bLightTrigger1 := tpLightTrig1.Q;
		MCU.typOUT.bLightTrigger2 := tpLightTrig2.Q;
		MCU.typOUT.bLightTrigger3 := tpLightTrig3.Q;
		MCU.typOUT.bLightTrigger4 := tpLightTrig4.Q;

		//Set outputs for camera's.
		MCU.typOUT.bCamTrigger1 := tpCamTrig1.Q;
		MCU.typOUT.bCamTrigger2 := tpCamTrig2.Q;
		MCU.typOUT.bCamTrigger3 := tpCamTrig3.Q;
		MCU.typOUT.bCamTrigger4 := tpCamTrig4.Q;
	END_IF

END_PROGRAM
```

#### Main.var - Local variables
```iecst
(********************************************************************
 * COPYRIGHT --
 ********************************************************************
 * Program: Main
 * File: Main.var
 * Author: jorkes
 * Created: August 14, 2014
 ********************************************************************
 * Local variables of program Main
 ********************************************************************)
VAR
	tonStart : TON;
	tonJogDelay : TON;
	tonBuzzerReset : TON;
	bRunRequest : BOOL := FALSE;
	srJogDelay : SR;
	TestPuls : PulsGenerator;
	iSpeed : INT := 1500; (*/30 = Hz (50)*)
	Var1 : USINT := 0;
	write : BOOL := FALSE;
	read : BOOL := FALSE;
	iBUEnabledMask : INT := -1;
	iMask : INT;
	iOut : INT;
	i : USINT; (*Loop*)
END_VAR
(*Variables for manual Camtrigger*)
VAR
	tiCamPuls : TIME := T#10ms;
	tiLightPuls : TIME := T#30ms;
	tpCamTrig1 : TP;
	tpCamTrig2 : TP;
	tpCamTrig3 : TP;
	tpCamTrig4 : TP;
	tpLightTrig1 : TP;
	tpLightTrig2 : TP;
	tpLightTrig3 : TP;
	tpLightTrig4 : TP;
END_VAR
```

#### MainInit.st
```iecst
(********************************************************************
 * COPYRIGHT --
 ********************************************************************
 * Program: Main
 * File: MainInit.st
 * Author: jorkes
 * Created: October 03, 2014
 *******************************************************************)

PROGRAM _INIT
	MCU.typInterface.bEnabled := TRUE;
END_PROGRAM
```

### Package Logical/MainBeltUnit - Package

### Program Logical/MainBeltUnit/BeltControl (IEC) - Program

#### BeltControl.st - Implementation code
```iecst
(********************************************************************
 * COPYRIGHT -- Microsoft
 ********************************************************************
 * Program: BeltControl
 * File: BeltControl.st
 * Author: jorkes
 * Created: November 28, 2014
 ********************************************************************
 * Implementation of program BeltControl
 ********************************************************************)

PROGRAM _INIT
	BeltSize := SIZEOF(	MBU.typInterface.bBeltShiftReg)/SIZEOF(	MBU.typInterface.bBeltShiftReg[idx]);
	MBU.typInterface.Command := MBU_CMD_INIT;
END_PROGRAM

PROGRAM _CYCLIC
	//Shift bunchbelt after beltsensor puls
	fbShiftBelt(MBU, EDGEPOS(SensControl_0.Q));

	//======================================
	//Reading sensors main belt
	//======================================

	//Vakkenband
	SensControl_0(IN := MBU.in_bMainBeltSensor1, tiSensDelay := MBU.typInterface.tiSensDelay1, tiSensPuls := MBU.typInterface.tiSensPuls);
	//Sponsband
	SensControl_1(IN := MBU.in_bMainBeltSensor2, tiSensDelay := MBU.typInterface.tiSensDelay2, tiSensPuls := MBU.typInterface.tiSensPuls);

	//After sensor puls do
	BindControl_0.IN := fbHasFlowersOnIndex(MBU,MBU.typInterface.usBindPos1) AND EDGEPOS(SensControl_0.Q); //MBU.typInterface.bBeltShiftReg[MBU.typInterface.usBindPos1];
	BindControl_1.IN := fbHasFlowersOnIndex(MBU,MBU.typInterface.usBindPos2) AND EDGEPOS(SensControl_0.Q); // MBU.typInterface.bBeltShiftReg[MBU.typInterface.usBindPos2];
	BufferControl.IN := fbHasFlowersOnIndex(MBU,MBU.typInterface.usAflegPos) AND EDGEPOS(SensControl_0.Q); //MBU.typInterface.bBeltShiftReg[MBU.typInterface.usAflegPos];
	KnifeControl.IN := fbHasFlowersOnIndex(MBU,MBU.typInterface.usKnifePos) AND EDGEPOS(SensControl_0.Q); //MBU.typInterface.bBeltShiftReg[MBU.typInterface.usKnifePos];

	IF EDGEPOS(MBU.typInterface.bEnable) AND MBU.typInterface.bEnable THEN
		MBU.typInterface.Command := MBU_CMD_INIT;
	END_IF

	// Log test van RONSPA
	//	IF EDGENEG(MBU.typInterface.bSimulate) THEN
	//		AsArLogWrite_1(enable := TRUE, ident := arlogBASE_USER_LOG_IDENT, logLevel := 1, errornr := 50000, mem := 0, len := 0, asciiString := ADR('MBU simulation OFF') );
	//		//UserLogEvent := TRUE;
	//	END_IF
	//
	//	IF EDGEPOS(MBU.typInterface.bSimulate) THEN
	//		AsArLogWrite_0(enable := TRUE, ident := arlogBASE_USER_LOG_IDENT, logLevel := 1, errornr := 50001, mem := 0, len := 0, asciiString := ADR('MBU simulation on') );
	//		//UserLogEvent := TRUE;
	//	END_IF

	IF MBU.typInterface.bEnable AND NOT MBU.typInterface.bSimulate THEN
		CASE MBU.typInterface.Command OF
			//======================================
			MBU_CMD_INIT:
				//======================================
				//MBU state
				MBU.typInterface.State := MBU_ST_INIT;

				//Inverter Motor 1
				//Vakkenband
				iSpeed1 := 690; //(23Hz)
				bRunReverse1 := FALSE;

				//Inverter Motor 2
				//Sponsband
				iSpeed2 := 670; //(22.3Hz)
				bRunReverse2 := FALSE;

				//Knife Motor
				iSpeed3 := 300;	//(10Hz)
				bRunReverse3 := FALSE;

				//Buffer Motor
				iSpeed4 := 600; //(20Hz)
				bRunReverse4 := FALSE;

				//Clear shiftregister bunchbelt
				FOR idx := 0 TO BeltSize - 1 DO
					fbSetFlowersOnIndex(MBU, idx, FALSE);  //		MBU.typInterface.bBeltShiftReg[idx] := FALSE;
				END_FOR

				//Check if frequency drive is Ready
				IF NOT( (MBU.motBelt1.InverterState_ = INV_ST_READY) OR (MBU.motBelt2.InverterState_ = INV_ST_READY) ) THEN// OR (MBU.motKnifeUnit.InverterState_ = INV_ST_READY) OR (MBU.motBufferBelt.InverterState_ = INV_ST_READY) )THEN
					MBU.typInterface.Command := MBU_CMD_STOP;
				ELSE
					MBU.typInterface.Command := MBU_CMD_RUN;
				END_IF

			//======================================
			MBU_CMD_RUN:
				//======================================
				tiActual := clock_ms();

				CASE ST_BELT OF
					//------------------------------------------------------
					CMD_WAIT:	//Check usMovePositions, if not NULL then move belt.
						//------------------------------------------------------
						IF (MBU.typInterface.usMovePositions <> 0) AND NOT(fbCheckBUReadyForDrop(BU, BUCount)) THEN
							MBU.typInterface.State := MBU_ST_RUN;
							MBU.typInterface.bReadyToReceive := FALSE;

							bRun1 := TRUE;	//Vakkenband
							bRun2 := TRUE;  //Sponsband

							//Sla tijd op zodra de bosband(en) start(en).
							tiStart1 := clock_ms();
							tiStart2 := tiStart1;
							ST_BELT := CMD_MOVE;
						END_IF
					//------------------------------------------------------
					CMD_MOVE:  //Move belt x positions
						//------------------------------------------------------
						IF (MBU.typInterface.usMovePositions < 1) THEN

							//Vakkenband
							IF EDGEPOS(SensControl_0.Q) THEN
								IF bSensCheck0 THEN
									MBU.typInterface.Command := MBU_CMD_FAULT;
								END_IF
								bSensCheck0 := TRUE;
								tiStop1 := clock_ms();
								tiDiff1[idx_Diff1] := tiStop1 - tiStart1;
								idx_Diff1 := (idx_Diff1 + 1) MOD 10;
							END_IF

							//Sponsband
							IF EDGEPOS(SensControl_1.Q) THEN
								IF bSensCheck1 THEN
									MBU.typInterface.Command := MBU_CMD_FAULT;
								END_IF
								bSensCheck1 := TRUE;
								tiStop2 := clock_ms();
								tiDiff2[idx_Diff2] := tiStop2 - tiStart2;
								idx_Diff2 := (idx_Diff2 + 1) MOD 10;
							END_IF

							IF bSensCheck0 AND bSensCheck1 THEN
								MBU.typInterface.usMovePositions := MBU.typInterface.usMovePositions - 1;
								bSensCheck0 := FALSE;
								bSensCheck1 := FALSE;
							END_IF
						ELSE
							ST_BELT := CMD_STOP;
						END_IF
					//------------------------------------------------------
					CMD_STOP:	//Wait for belt triggers
						//------------------------------------------------------

						//Vakkenband
						IF EDGEPOS(SensControl_0.Q) THEN
							bRun1 := FALSE;
							tiStop1 := clock_ms();
							tiDiff1[idx_Diff1] := tiStop1 - tiStart1;
							idx_Diff1 := (idx_Diff1 + 1) MOD 10;
						END_IF

						//Sponsband
						IF EDGEPOS(SensControl_1.Q) THEN
							bRun2 := FALSE;
							tiStop2 := clock_ms();
							tiDiff2[idx_Diff2] := tiStop2 - tiStart2;
							idx_Diff2 := (idx_Diff2 + 1) MOD 10;
						END_IF

						//Wacht totdat motoren uitstaan en ga dan weer naar READY state.
						IF NOT(bRun1) AND NOT(bRun2) THEN
							MBU.typInterface.bReadyToReceive := TRUE;
							MBU.typInterface.State := MBU_ST_READY;
							MBU.typInterface.usMovePositions := MBU.typInterface.usMovePositions - 1;
							ST_BELT := CMD_WAIT;
						END_IF
				END_CASE

			//======================================
			MBU_CMD_STOP:
			//======================================

			//======================================
			MBU_CMD_MANUAL:
			//======================================

			//======================================
			MBU_CMD_FAULT:
			//======================================
				MBU.typInterface.bFault := TRUE;
				bRun1 := FALSE;
				bRun2 := FALSE;
				MBU.typInterface.State := MBU_ST_ERROR;
		END_CASE

	ELSIF MBU.typInterface.bReset THEN
		//freq. regelaaars
		MBU.typInterface.bReset := FALSE;
		MBU.typInterface.Command := MBU_CMD_RUN; // Init gooit de buffers leeg.

	ELSIF MBU.typInterface.bSimulate THEN
		MBU.typInterface.State := MBU_ST_SIMULATED;
	ELSE
		MBU.typInterface.State := MBU_ST_DISABLED;
	END_IF

	//Call function blocks
	BindControl_1(tiSensDelay := MBU.typInterface.tiBindDelay2, tiSensPuls := MBU.typInterface.tiBindPuls);
	BindControl_0(tiSensDelay := MBU.typInterface.tiBindDelay1, tiSensPuls := MBU.typInterface.tiBindPuls);
	BufferControl(tiSensDelay := MBU.typInterface.tiBufferDelay, tiSensPuls := MBU.typInterface.tiBufferPuls);
	KnifeControl(tiSensDelay := T#1ms, tiSensPuls := MBU.typInterface.tiKnifePuls);

	//======================================
	//Outputs for binders
	//======================================
	MBU.out_bBinder1 := BindControl_0.Q;
	MBU.out_bBinder2 := BindControl_1.Q;
	bRun3 := KnifeControl.Q;
	bRun4 := BufferControl.Q;

	//======================================
	//Countup index of shiftregister bunchbelt
	//======================================
	IF EDGEPOS(SensControl_0.Q) OR MBU.typInterface.bSimulate THEN
		idxBeltPos := (idxBeltPos + 1) MOD MBU.typInterface.usBunchPositions;
	END_IF

	//======================================
	//Motor BeltControl 1
	//Vakkenband
	//======================================
	MBU.motBelt1.bRun := bRun1 OR MBU.typInterface.bToggleBelt;
	MBU.motBelt1.bRunReverse := FALSE;
	MBU.motBelt1.bResetFault := MBU.typInterface.bReset;
	MBU.motBelt1.iSpeed := iSpeed1;
	MBU.motBelt1(MotorStruc := MBU.typBeltMotor1);

	//======================================
	//Motor BeltControl 2
	//Sponsband
	//======================================
	MBU.motBelt2.bRun := bRun2 OR MBU.typInterface.bToggleBelt;
	MBU.motBelt2.bRunReverse := FALSE;
	MBU.motBelt2.bResetFault := MBU.typInterface.bReset;
	MBU.motBelt2.iSpeed := iSpeed2;
	MBU.motBelt2(MotorStruc := MBU.typBeltMotor2);

	//======================================
	//Motor Knife
	//======================================
	MBU.motKnifeUnit.bRun := bRun3 OR MBU.typInterface.bToggleKnife OR MBU.typInterface.bToggleBelt; //bToggleBelt just for test JORKES
	MBU.motKnifeUnit.bRunReverse := FALSE;
	MBU.motKnifeUnit.bResetFault := MBU.typInterface.bReset;
	MBU.motKnifeUnit.iSpeed := iSpeed3;
	MBU.motKnifeUnit(MotorStruc := MBU.typKnifeUnit);

	//======================================
	//Motor Bufferbelt
	//======================================
	MBU.motBufferBelt.bRun := bRun4 OR MBU.typInterface.bToggleBuffer OR MBU.typInterface.bToggleBelt; //bToggleBelt just for test JORKES
	MBU.motBufferBelt.bRunReverse := FALSE;
	MBU.motBufferBelt.bResetFault := MBU.typInterface.bReset;
	MBU.motBufferBelt.iSpeed := iSpeed4;
	MBU.motBufferBelt(MotorStruc := MBU.typBufferMotor);

	// MBU State
	MBU.typInterface.bFault := MBU.typBeltMotor1.status.bFault OR
	MBU.typBeltMotor2.status.bFault OR
	MBU.typBufferMotor.status.bFault OR
	MBU.typKnifeUnit.status.bFault OR
	MBU.typInterface.bSimulate;
END_PROGRAM
```

#### BeltControl.typ - Local data types
```iecst
(********************************************************************
 * COPYRIGHT -- Microsoft
 ********************************************************************
 * Program: BeltControl
 * File: BeltControl.typ
 * Author: jorkes
 * Created: November 28, 2014
 ********************************************************************
 * Local data types of program BeltControl
 ********************************************************************)

TYPE
	InterfaceMBU : 	STRUCT
		bEnabled : BOOL; (*Enable MBU*)
	END_STRUCT;
	MainBeltControl : 	STRUCT
		typeInterface : InterfaceMBU;
	END_STRUCT;
END_TYPE
```

#### BeltControl.var - Local variables
```iecst
(********************************************************************
 * COPYRIGHT -- Microsoft
 ********************************************************************
 * Program: BeltControl
 * File: BeltControl.var
 * Author: jorkes
 * Created: November 28, 2014
 ********************************************************************
 * Local variables of program BeltControl
 ********************************************************************)
(*check time between belt positions*)
VAR
	idx_Diff2 : USINT;
	idx_Diff1 : USINT;
	tiActual : TIME;
	tiDiff2 : ARRAY[0..9] OF TIME;
	tiStop2 : TIME;
	tiStart2 : TIME;
	tiDiff1 : ARRAY[0..9] OF TIME;
	tiStop1 : TIME;
	tiStart1 : TIME;
END_VAR
(*State machine beltcontrol*)
VAR
	bSensCheck1 : BOOL;
	bSensCheck0 : BOOL;
	ST_BELT : USINT := 0;
END_VAR
VAR CONSTANT
	CMD_WAIT : USINT := 0;
	CMD_STOP : USINT := 2;
	CMD_MOVE : USINT := 1;
END_VAR
VAR
	BeltSize : USINT := 0;
	idxBeltPos : USINT := 0;
	bTest : BOOL;
	idx : USINT := 0;
END_VAR
(*Inverters*)
VAR
	InverterCommand : enumINV_CMD;
	InverterState : enumINV_ST;
END_VAR
(*Beltmotor1 - Vakkenband*)
VAR
	bRun1 : BOOL;
	bRunReverse1 : BOOL;
	bResetFault1 : BOOL;
	iSpeed1 : INT := 690; (*23Hz*)
END_VAR
(*Beltmotor2 - Sponsband*)
VAR
	bRun2 : BOOL;
	bRunReverse2 : BOOL;
	bResetFault2 : BOOL;
	iSpeed2 : INT := 670; (*22.3Hz*)
END_VAR
(*Knifemotor*)
VAR
	bRun3 : BOOL;
	bRunReverse3 : BOOL;
	bResetFault3 : BOOL;
	iSpeed3 : INT := 20; (*20Hz*)
END_VAR
(*Buffermotor*)
VAR
	bRun4 : BOOL;
	bRunReverse4 : BOOL;
	bResetFault4 : BOOL;
	iSpeed4 : INT := 20; (*20Hz*)
END_VAR
(*Sensor checks*)
VAR
	KnifeControl : fbSensDelay;
	BufferControl : fbSensDelay;
	BindControl_1 : fbSensDelay;
	BindControl_0 : fbSensDelay;
	SensControl_1 : fbSensDelay;
	SensControl_0 : fbSensDelay;
	AsArLogWrite_1 : AsArLogWrite := (0);
	AsArLogWrite_0 : AsArLogWrite := (0);
END_VAR
```

### Package Logical/BunchUnits - Package

### Program Logical/BunchUnits/BU_Ref (IEC) - Bunch Unit Ref (BU)

#### BunchUnit.st - Implementation code
```iecst
PROGRAM _CYCLIC

	//=========================================Program=====================================================
	//Always check if BunchUnit is enabled, daarna controleren of de bosunit is geïnitialiseerd.
	//Zo ja, dan mag het de 'run' cyclus beginnen, zo niet dan wordt eerst het initialisatie proces gestart.
	BU[i].typOUT.bEnableServo := BU[i].typOUT.bStopServo AND BU[i].typInterface.bEnable AND NOT BU[i].typInterface.bReset;
	BU[i].typOUT.bStopServo := BU[i].typInterface.bEnable;
	BU[i].typOUT.bEndStageServo := BU[i].typInterface.bEnable;

	IF BU[i].typInterface.bReset THEN
		ServoReset(BU[i]);
		BU[i].bAddFlower := FALSE;
		BU[i].bBusyDrop := FALSE;
		BU[i].GripperControl.IN := FALSE;

		IF BU[i].typInterface.Status = BU_ST_FAILURE THEN
			BU[i].typInterface.Command := BU_CMD_Init;
		END_IF
		//Reset fault
		IF NOT BU[i].typBunchBelts.status.bFault THEN
			bResetFault := TRUE;
		ELSE
			bResetFault := TRUE;
		END_IF
		// BU[i].typInterface.bReset := FALSE;
	ELSE
		bResetFault := FALSE;
		IF EDGEPOS( BU[i].typInterface.bSimulation ) THEN
			BU[i].typInterface.bEnable := TRUE;
			BU[i].typInterface.Status := BU_ST_RECEIVE;
			BU[i].typInterface.Command := BU_CMD_Receive;
		END_IF
		IF NOT BU[i].typInterface.bEnable THEN
			BU[i].typInterface.Status := BU_ST_DISABLED;
			BU[i].typInterface.bManualCmd := FALSE;
			bRun := FALSE;
		ELSE
			IF EDGEPOS(BU[i].typInterface.bManualCmd) THEN
				// Remove old cmd's
				BU[i].typInterface.bManualUpCmd := FALSE;
				BU[i].typInterface.bManualDownCmd := FALSE;
			END_IF

			IF  BU[i].typInterface.bManualCmd THEN
				BU[i].typInterface.Status := BU_ST_MANUAL;
				BU[i].typInterface.Command := BU_CMD_Manual;
			END_IF
			//==================================
			//Check for initialisation commando.
			//==================================

			IF BU[i].typInterface.Status = BU_ST_DISABLED THEN
				BU[i].typInterface.Command := BU_CMD_Init;
			END_IF

			//==================================
			//BunchUnit initialisation
			//==================================

			CASE BU[i].typInterface.Command OF
				//==================================
				BU_CMD_Init: // 1
				//==================================
					//Init freq. inverter bunchbelt
					//Default speed
					BU[i].typInterface.iSpeedBunchbelt := 2700; //(90Hz)
					//Direction setting
					bRunReverse := FALSE;

					//FOR TESTING PURPOSES (*TESTING*) 17-12-2014
					out_bModule1[0] := TRUE;
					out_bModule1[1] := TRUE;

					//Set al pneumatics to default situation.
					BU[i].typOUT.bActivateGripper := FALSE;
					BU[i].typOUT.bBunchGripper := FALSE;

					Elevator(BU[i], BU_ELEVATOR_UP);
					BU[i].typInterface.Command := BU_CMD_Home;
					BU[i].typInterface.Status := BU_ST_INIT;
				//==================================
				BU_CMD_Ready: // 6
				//==================================
					BU[i].typInterface.Status := BU_ST_RETURN;
					IF BU[i].typOUT.bBunchGripper THEN
						BU[i].typOUT.bBunchGripper := FALSE;
					END_IF

					IF NOT BU[i].typIN.bElevatorUp THEN
						Elevator(BU[i], BU_ELEVATOR_UP);
					ELSE
						//When elevator up, close releasegrippers
						BU[i].typOUT.bReleaseGripper := FALSE;
					END_IF

					IF BU[i].typIN.bElevatorMid OR BU[i].typIN.bElevatorUp THEN
						BU[i].typInterface.iReceivePos := Settings.iBUIdealReceivePosition;
						ServoMovePosition(BU[i],  BU[i].typInterface.iReceivePos, BU[i].typInterface.usServoSpeed); //  BU[i].typeSettings.iReceivePos +
						//Bunchbelt release
						BU[i].typInterface.bReadyForDrop := FALSE;
						bRun := FALSE;
					END_IF

					IF BU[i].typServo.status.SPOS.bMC AND BU[i].typIN.bElevatorUp THEN
						BU[i].typInterface.Command := BU_CMD_Receive;
						// The loop is completed, now the active BIT can be reset.
						BU[i].bAddFlower := FALSE;
						BU[i].bBusyDrop := FALSE;
					END_IF
				//==================================
				BU_CMD_Home: // 2
				//==================================
					//Check of elevator is in upper position.
					IF BU[i].typIN.bElevatorUp THEN

						IF NOT BU[i].typServo.status.SPOS.bREF THEN
							//Homing servo.
							IF NOT ServoHome(BU[i]) THEN
								BU[i].typInterface.bFault := TRUE;
							END_IF
							//Check for homing complete signal.
						ELSE
							//Put usInitState to rest(99) and set usState to active(0).
							BU[i].typInterface.Status := BU_ST_HOME;
							//BU[i].typInterface.Command := BU_CMD_Drop;
							BU[i].typInterface.Command := BU_CMD_Ready;
						END_IF
					END_IF
				//==================================
				BU_CMD_Receive: // 3
				//==================================
					//Check if frequency drive is Ready
					IF NOT BU[i].typIN.bElevatorUp  AND NOT BU[i].typInterface.bSimulation THEN
						Elevator(ThisBU := BU[i], BU_ELEVATOR_UP);
						BU[i].typInterface.Status := BU_ST_MOVE_ELEVATOR_UP;
					ELSE
						ServoMovePosition(BU[i],  BU[i].typInterface.iReceivePos, BU[i].typInterface.usServoSpeed);

						// ***********************************************
						// Manual add flower!!! TEST RSPA
						IF BU[i].typInterface.bAddFlowerNow THEN
							BU[i].typInterface.bAddFlowerNow := FALSE;
							SHFTREG.typGripper[usGripperIndex].usSetTarget := INT_TO_SINT(i);
							//SHFTREG.typGripper[usGripperIndex].uiTimingBU16 := 4;
						//	IF BU[i].typInterface.bEmptyCmd THEN
								SHFTREG.typGripper[usGripperIndex].siEmptyBU := INT_TO_SINT(i);
						//	END_IF
							SHFTREG.typGripper[usGripperIndex].uiCorrection := testPosition;
							// Release the Reject
							SHFTREG.typGripper[usGripperIndex].bRejectActive := TRUE;
							SHFTREG.typGripper[usGripperIndex].bRejectOnOff := FALSE;

							// Activate the Reject
							SHFTREG.typGripper[(usGripperIndex + 1)  MOD  SHFTREG.uiGripperCnt].bRejectActive := TRUE;
							SHFTREG.typGripper[(usGripperIndex + 1)  MOD  SHFTREG.uiGripperCnt].bRejectOnOff := TRUE;

							//SHFTREG.typGripANDper[0].uiTimingBU16
						END_IF
						// ***********************************************

						usGripperIndex := ( SHFTREG.typCounters.usChainCounter  ) MOD  SHFTREG.uiGripperCnt; //  + BU[i].usChainPos + RU.usChainPos  + RU.usChainPos

						// BunchBeltControl.Q is SET by the Shift register
						BU[i].BunchBeltControl(IN := BU[i].GripperControl.Q, PT := INT_TO_TIME( Settings.BU_BunchBeltTime)); // T#400ms);
						bRun := BU[i].BunchBeltControl.Q;
						IF EDGENEG(BU[i].BunchBeltControl.Q) THEN // The flower was added
							//Counting stems in bunchunit
							BU[i].typInterface.usStemCount := BU[i].typInterface.usStemCount + 1;
							// BU[i].bAddFlower := FALSE; Wordt al gedaan in shift register....
						END_IF

						// Move to receive position  AND (BU[i].motBunchBelts.InverterState_ = INV_ST_READY)
						IF BU[i].typServo.status.SPOS.bMC OR  BU[i].typInterface.bSimulation THEN
							BU[i].typInterface.Status := BU_ST_RECEIVE;
						ELSIF NOT(BU[i].motBunchBelts.InverterState_ = INV_ST_READY) AND NOT BU[i].typInterface.bSimulation THEN
							BU[i].typInterface.Command := BU_CMD_Hold;
						ELSE
							BU[i].typInterface.Status := BU_ST_RECEIVE_POS;
						END_IF
						//						// Check for next gripper
						//						IF EDGEPOS( SHFTREG.typCounters.usChainCounter) THEN
						//							//
						//							usGripperIndex = ( SHFTREG.typCounters.usChainCounter + SHFTREG.uiGripperCnt - BU[i].usChainPos) MOD  SHFTREG.uiGripperCnt;
						//							IF( SHFTREG.typGripper[usGripperIndex].usSetTarget == i)
						//								// Start timer
//							END_IF
						//						END_IF

						IF NOT BU[i].bAddFlower AND NOT bRun AND NOT(BU[i].typInterface.Status = BU_ST_RECEIVE_POS) THEN
							// Check if must empty
							IF 	BU[i].typInterface.bEmptyCmd THEN
								BU[i].typInterface.bEmptyCmd := FALSE;
								IF NOT BU[i].typInterface.bSimulation THEN
									BU[i].bBusyDrop := TRUE;
									BU[i].typInterface.Command := BU_CMD_Drop;
								ELSE
									BU[i].bBusyDrop := FALSE;
								END_IF
							END_IF
						END_IF
					END_IF
				//==================================
				BU_CMD_Drop: // 4
				//==================================
					//Bunchbelt lock
					BU[i].typInterface.bReadyForDrop := TRUE;
					MBU.typInterface.bReadyToReceive := TRUE;  // TEST SHOULD BE FROM MCU!!!!!!!!!
					BU[i].typInterface.usStemCount := 0;

					tonDropDelay.PT := BU[i].typSettings.tiDropDelay;
					IF BU[i].typIN.bElevatorUp THEN // AND NOT BU[i].typInterface.bSimulation THEN
						ServoMovePosition(BU[i], BU[i].typInterface.iReleasePos,  BU[i].typSettings.usSpeed);
						BU[i].typInterface.Status := BU_ST_DROP_POS;

						// AND ABS( BU[i].typInterface.iReleasePos - BU[i].Servo.status.VAL2.diPosition ) < 5
						IF (BU[i].typServo.status.SPOS.bMC  AND ABS( BU[i].typInterface.iReleasePos - BU[i].typServo.status.VAL2.diPosition ) < 5) OR  BU[i].typInterface.bSimulation THEN
							BU[i].typInterface.Status := BU_ST_WAIT_MCU;
							IF  MBU.typInterface.bReadyToReceive OR  BU[i].typInterface.bSimulation THEN
								//Check for current position. When safe, activate elevator down. Check bunchbelt is ready to receive bunch.
								Elevator(BU[i], BU_ELEVATOR_DOWN);
								BU[i].typOUT.bBunchGripper := TRUE;
								BU[i].typInterface.Status := BU_ST_MOVE_ELEVATOR_DOWN;
								BU[i].typInterface.usStemCount := 0;
							END_IF
						END_IF
					ELSE
						// Fase 2 of drop lowering Elevator
						IF BU[i].typIN.bElevatorDown THEN
							// Ready to drop
							BU[i].typOUT.bReleaseGripper := TRUE;
							bRun := TRUE;
							tonDropDelay.IN := TRUE;
							tonDropDelay();
							BU[i].typInterface.Status := BU_ST_RELEASING;

							IF tonDropDelay.Q THEN
								tonDropDelay.IN := FALSE;
								BU[i].typOUT.bBunchGripper := TRUE;
								BU[i].typInterface.Status := BU_ST_DROPPED;
								BU[i].typInterface.Command := BU_CMD_DropReady;

								//JORKES 25-02-2015
								//Put flowers into shiftregister bunchbelt.
								//MBU.typInterface.bBeltShiftReg[BU[i].typSettings.usBunchBeltPosition] := TRUE;
								fbSetFlowersOnIndex(MBU, BU[i].typSettings.usBunchBeltPosition, TRUE );
							END_IF
						END_IF
					END_IF
				//==================================
				BU_CMD_DropReady: // 5
				//==================================
					tonDropReadyDelay.PT := BU[i].typSettings.tiDropReadyDelay;
					tonDropReadyDelay();
					tonDropReadyDelay.IN := TRUE;

					IF tonDropReadyDelay.Q THEN
						tonDropReadyDelay.IN := FALSE;
						BU[i].typInterface.Status := BU_ST_DROPPED;
						BU[i].typInterface.Command := BU_CMD_Ready;
					END_IF
				//==================================
				BU_CMD_Manual:
				//==================================
					IF NOT BU[i].typInterface.bManualCmd  THEN
						BU[i].typInterface.Command := BU_CMD_Init;
					ELSE
						IF BU[i].typInterface.iManualPosition <> BU[i].typServo.command.PARA2.diPosition THEN
							ServoMovePosition(BU[i], BU[i].typInterface.iManualPosition,  BU[i].typInterface.usManualSpeed);
						END_IF
					END_IF
					IF  BU[i].typInterface.bManualUpCmd THEN
						BU[i].typInterface.bManualUpCmd := NOT (BU[i].typIN.bElevatorMid OR BU[i].typIN.bElevatorUp);
						Elevator(BU[i], BU_ELEVATOR_UP);
					END_IF
					IF  BU[i].typInterface.bManualDownCmd THEN
						BU[i].typInterface.bManualDownCmd := NOT (BU[i].typIN.bElevatorMid OR BU[i].typIN.bElevatorDown);
						Elevator(BU[i], BU_ELEVATOR_DOWN);
					END_IF

					IF BU[i].typInterface.bManualGripperCmd THEN
						BU[i].typOUT.bBunchGripper := TRUE;
						BU[i].typOUT.bActivateGripper := TRUE;
						BU[i].typOUT.bReleaseGripper := TRUE;
					ELSE
						BU[i].typOUT.bBunchGripper := FALSE;
						BU[i].typOUT.bActivateGripper := FALSE;
						BU[i].typOUT.bReleaseGripper := FALSE;
					END_IF
				//==================================
				BU_CMD_Hold:
				//==================================
					BU[i].typInterface.Status := BU_ST_FAILURE;
					bRun := FALSE;

			END_CASE
		END_IF
	END_IF

	//======================================
	//Motor Bunchbelt
	//======================================
	//Call function motorstruct
	BU[i].motBunchBelts.bRun := bRun OR BU[i].typInterface.bToggleBunchBelt;
	BU[i].motBunchBelts.bRunReverse := bRunReverse;
	BU[i].motBunchBelts.bResetFault := bResetFault;
	BU[i].motBunchBelts.iSpeed := BU[i].typInterface.iSpeedBunchbelt;
	BU[i].motBunchBelts(MotorStruc := BU[i].typBunchBelts);

	IF EDGEPOS(BU[i].typIN.bPosMove) THEN
		ServoMovePosition(BU[i],DINT_TO_INT( BU[i].typServo.command.PARA2.diPosition + 50), BU[i].typSettings.usHomeSpeed);
	END_IF

	IF EDGEPOS (BU[i].typIN.bNegMove) THEN
		ServoMovePosition(BU[i], DINT_TO_INT(BU[i].typServo.command.PARA2.diPosition - 50), BU[i].typSettings.usHomeSpeed);
	END_IF

	BU[i].typInterface.Status := CheckTimers(BU[i], BU[i].typInterface.Status);

	// Fault status for GUI
	BU[i].typInterface.bFault := NOT BU[i].typBunchBelts.packed.ModuleOk OR
									NOT BU[i].typServo.bOnLine OR
									NOT BU[i - (i MOD 2)].typIN.bOnline OR
									NOT BU[i - (i MOD 2)].typOUT.bOnline OR
									BU[i].typInterface.bManualCmd OR
									NOT BU[i].typInterface.bEnable OR
									BU[i].typInterface.Status = BU_ST_FAILURE;

	//==================================
	//Visualistion
	//==================================

	//ElevatorState
	IF BU[i].typIN.bElevatorDown THEN
		BU[i].typIN.ElevatorState := BU_VISU_ELEVATOR_DOWN;
	ELSIF BU[i].typIN.bElevatorMid THEN
		BU[i].typIN.ElevatorState := BU_VISU_ELEVATOR_MID;
	ELSIF BU[i].typIN.bElevatorUp THEN
		BU[i].typIN.ElevatorState := BU_VISU_ELEVATOR_UP;
	END_IF

	//ReleaseState
	IF BU[i].typOUT.bReleaseGripper THEN
		BU[i].typOUT.ReleaseState := BU_VISU_RELEASE_OUT;
	ELSE
		BU[i].typOUT.ReleaseState := BU_VISU_RELEASE_IN;;
	END_IF

	//GripperState
	IF BU[i].typOUT.bActivateGripper THEN
		BU[i].typOUT.GripperState := BU_VISU_GRIPPER_OUT;
	ELSE
		BU[i].typOUT.GripperState := BU_VISU_GRIPPER_IN;
	END_IF

END_PROGRAM
```

#### BunchUnit.var - Local variables
```iecst
(********************************************************************
 * COPYRIGHT --
 ********************************************************************
 * Program: BU
 * File: BU.var
 * Author: ronspa
 * Created: September 25, 2014
 ********************************************************************
 * Local variables of program BU
 ********************************************************************)
VAR
	testPosition : UINT := 400;
	i : INT; (*Bos Unit index*)
	tonLift : TON;
	tonDropReadyDelay : TON; (*Delay when released*)
	tonDropDelay : TON; (*Delay of gripper afther drop*)
	tpBunchBelts : TP;
	tpResetInv : TP;
	_BunchBeltControl : fbSensControl;
	_GripperControl : fbSensControl;
	usGripperIndex : USINT;
END_VAR
(*FreqInverter control*)
VAR
	bRun : BOOL;
	bRunReverse : BOOL := FALSE;
	bResetFault : BOOL;
	PulsGenerator_0 : PulsGenerator;
END_VAR
```

### Program Logical/BunchUnits/SC_Ref (IEC) - Servo Control Ref (SC)

#### SC.st - Implementation code
```iecst
(********************************************************************
 * COPYRIGHT --
 ********************************************************************
 * Program: ServoControl
 * File: ServoControl.st
 * Author: jorkes
 * Created: July 30, 2014
 ********************************************************************
 * Implementation of program ServoControl
 ********************************************************************)

PROGRAM _CYCLIC
	//=========================================Servo variables===========================================

	//Write back to CPOS
	BU[i].typServo.command.CPOS.bHALT := FALSE;
	BU[i].typServo.command.CPOS.bSTART := FALSE;
	BU[i].typServo.command.CPOS.bHOM := FALSE;
	BU[i].typServo.command.CPOS.bJOGP := FALSE;
	BU[i].typServo.command.CPOS.bJOGN := FALSE;
	BU[i].typServo.command.CPOS.bTEACH := FALSE;
	BU[i].typServo.command.CPOS.bCLEAR := FALSE;
	BU[i].typServo.command.CPOS.bNU := FALSE;

	//Write back to CCON
	BU[i].typServo.command.CCON.bENABLE := FALSE;
	BU[i].typServo.command.CCON.bSTOP := FALSE;
	BU[i].typServo.command.CCON.bBRAKE := FALSE;
	BU[i].typServo.command.CCON.bRESET := FALSE;
	BU[i].typServo.command.CCON.bNU := FALSE;
	BU[i].typServo.command.CCON.bLOCK := FALSE;
	BU[i].typServo.command.CCON.bOPM1 := FALSE;
	BU[i].typServo.command.CCON.bOPM2 := FALSE;

	//Velocity in %
	BU[i].typServo.status.VAL1.usVelocity := BU[i].typServo.packed.VAL1;
	//Position
	BU[i].typServo.status.VAL2.diPosition := BU[i].typServo.packed.VAL2;

	BU[i].typServo.status.SPOS.uiSPOS 	:= BU[i].typServo.packed.SPOS AND 16#FF;	// Mask the SPOS status word
	BU[i].typServo.status.SPOS.bHALT 	:= BU[i].typServo.status.SPOS.uiSPOS.0;	// bit 0 = Halt
	BU[i].typServo.status.SPOS.bACK		:= BU[i].typServo.status.SPOS.uiSPOS.1;	// bit 1 = Acknowledge start
	BU[i].typServo.status.SPOS.bMC 		:= BU[i].typServo.status.SPOS.uiSPOS.2;	// bit 2 = Motion complete
	BU[i].typServo.status.SPOS.bTEACH	:= BU[i].typServo.status.SPOS.uiSPOS.3;	// bit 3 = Acknowledge teach/sampling
	BU[i].typServo.status.SPOS.bMOV		:= BU[i].typServo.status.SPOS.uiSPOS.4;	// bit 4 = Axis is moving
	BU[i].typServo.status.SPOS.bDEV		:= BU[i].typServo.status.SPOS.uiSPOS.5;	// bit 5 = Drag (deviation) error
	BU[i].typServo.status.SPOS.bSTILL	:= BU[i].typServo.status.SPOS.uiSPOS.6;	// bit 6 = Standstill control
	BU[i].typServo.status.SPOS.bREF		:= BU[i].typServo.status.SPOS.uiSPOS.7;	// bit 7 = Axis is referencend

	BU[i].typServo.status.SCON.uiSCON 	:= BU[i].typServo.packed.SCON AND 16#FF;	// Mask the SCON status word
	BU[i].typServo.status.SCON.bENABLED	:= BU[i].typServo.status.SCON.uiSCON.0;	// bit 0 = Drive enabled
	BU[i].typServo.status.SCON.bOPEN 	:= BU[i].typServo.status.SCON.uiSCON.1;	// bit 1 = Operation enabled
	BU[i].typServo.status.SCON.bWARN 	:= BU[i].typServo.status.SCON.uiSCON.2;	// bit 2 = Warning
	BU[i].typServo.status.SCON.bFAULT 	:= BU[i].typServo.status.SCON.uiSCON.3;	// bit 3 = Fault
	BU[i].typServo.status.SCON.b24VL 	:= BU[i].typServo.status.SCON.uiSCON.4;	// bit 4 = Supply voltage is applied
	BU[i].typServo.status.SCON.bLOCK 	:= BU[i].typServo.status.SCON.uiSCON.5;	// bit 5 = Drive control by software
	BU[i].typServo.status.SCON.bOPM1	:= BU[i].typServo.status.SCON.uiSCON.6;	// bit 6 = Display operating mode
	BU[i].typServo.status.SCON.bOPM2 	:= BU[i].typServo.status.SCON.uiSCON.7;	// bit 7 = Display operating mode

	//==================================
	//ServoControl
	//==================================

//	CASE BU[i].typServo.gCommand OF
	CASE BU[i].typServo.enumServoCmd OF
		SERVO_CMD_HOME:
			ControllerState := 10;
			IF BU[i].typServo.status.SCON.bENABLED AND BU[i].typServo.status.SCON.bOPEN AND BU[i].typServo.status.SCON.b24VL THEN
				IF BU[i].typServo.status.SPOS.bHALT THEN
					BU[i].typServo.command.CPOS.bHOM := TRUE;
				END_IF
			END_IF
			IF BU[i].typServo.status.SPOS.bREF THEN
				BU[i].typServo.enumServoCmd := SERVO_CMD_READY;
			END_IF
		SERVO_CMD_RUN:
			ControllerState := 10;
			IF BU[i].typServo.status.SPOS.bMC THEN
				CASE SetServo OF
					0:
						tiMusecStart := clock_ms();
						SetServo := 1;
					1:
						//Store stop time (us)
						tiMusecStop := clock_ms();
						tiMusecDiff := tiMusecStop - tiMusecStart;
						IF tiMusecDiff > T#100ms THEN
							//'Start position task'
							BU[i].typServo.command.CPOS.bSTART := 1;
							BU[i].typServo.enumServoCmd := SERVO_CMD_READY;
							SetServo := 0;
						END_IF
				END_CASE
			END_IF
		SERVO_CMD_RESET:
			BU[i].typServo.command.CCON.bRESET := TRUE;
			BU[i].typServo.enumServoCmd := SERVO_CMD_READY;
		SERVO_CMD_READY:
			// Ready to receive new command
	END_CASE

	//==================================
	//State
	//==================================

	CASE ControllerState OF
		10:	//CCON
			BU[i].typServo.command.CCON.bENABLE := TRUE;
			BU[i].typServo.command.CCON.bSTOP := TRUE;
			BU[i].typServo.command.CCON.bOPM1 := TRUE;
			//CPOS
			BU[i].typServo.command.CPOS.bHALT := TRUE;
	END_CASE

	IF BU[i].typServo.status.SPOS.bREF THEN
		IF BU[i].typServo.status.SPOS.bMOV THEN
			BU[i].typServo.enumServoState := SERVO_RUNNING;
		ELSE
			BU[i].typServo.enumServoState := SERVO_READY;
		END_IF
	ELSIF NOT BU[i].typServo.status.SPOS.bREF THEN
		IF BU[i].typServo.status.SPOS.bMOV THEN
			BU[i].typServo.enumServoState := SERVO_IS_HOMING;
		ELSE
			BU[i].typServo.enumServoState := SERVO_HOMING_NOT_COMPLETED;
		END_IF
	END_IF
	IF NOT BU[i].typServo.status.SCON.bENABLED THEN
		BU[i].typServo.enumServoState := SERVO_DISABLED;
	END_IF
	IF BU[i].typServo.status.SCON.bFAULT THEN
		BU[i].typServo.enumServoState := SERVO_FAULT;
	END_IF

	//Write back to CPOS
	BU[i].typServo.packed.CPOS.0 := BU[i].typServo.command.CPOS.bHALT;
	BU[i].typServo.packed.CPOS.1 := BU[i].typServo.command.CPOS.bSTART;
	BU[i].typServo.packed.CPOS.2 := BU[i].typServo.command.CPOS.bHOM;
	BU[i].typServo.packed.CPOS.3 := BU[i].typServo.command.CPOS.bJOGP;
	BU[i].typServo.packed.CPOS.4 := BU[i].typServo.command.CPOS.bJOGN;
	BU[i].typServo.packed.CPOS.5 := BU[i].typServo.command.CPOS.bTEACH;
	BU[i].typServo.packed.CPOS.6 := BU[i].typServo.command.CPOS.bCLEAR;
	BU[i].typServo.packed.CPOS.7 := BU[i].typServo.command.CPOS.bNU;

	//Write back to CCON
	BU[i].typServo.packed.CCON.0 := BU[i].typServo.command.CCON.bENABLE;
	BU[i].typServo.packed.CCON.1 := BU[i].typServo.command.CCON.bSTOP;
	BU[i].typServo.packed.CCON.2 := BU[i].typServo.command.CCON.bBRAKE;
	BU[i].typServo.packed.CCON.3 := BU[i].typServo.command.CCON.bRESET;
	BU[i].typServo.packed.CCON.4 := BU[i].typServo.command.CCON.bNU;
	BU[i].typServo.packed.CCON.5 := BU[i].typServo.command.CCON.bLOCK;
	BU[i].typServo.packed.CCON.6 := BU[i].typServo.command.CCON.bOPM1;
	BU[i].typServo.packed.CCON.7 := BU[i].typServo.command.CCON.bOPM2;

	//Write back to PARA1 and PARA2
	BU[i].typServo.packed.PARA1 := BU[i].typServo.command.PARA1.usVelocity;
	BU[i].typServo.packed.PARA2 := BU[i].typServo.command.PARA2.diPosition;

END_PROGRAM
```

#### SC.var - Local variables
```iecst
(********************************************************************
 * COPYRIGHT --
 ********************************************************************
 * Program: ServoControl
 * File: ServoControl.var
 * Author: jorkes
 * Created: July 30, 2014
 ********************************************************************
 * Local variables of program ServoControl
 ********************************************************************)
VAR
	NewServoPos : USINT;
	tiMusecDiff : TIME;
	tiMusecStop : TIME;
	tiMusecStart : TIME;
	ServoState : SERVO_Status_enum;
	ControllerState : INT;
	SetServo : INT;
	i : USINT;
END_VAR
```

### Program Logical/BunchUnits/Init (IEC) - Init setting for Bunch units

#### Init.st - Initialization code
```iecst
(********************************************************************
 * COPYRIGHT --
 ********************************************************************
 * Program: InitSettings
 * File: InitSettingsInit.st
 * Author: jorkes
 * Created: October 03, 2014
 ********************************************************************
 * Implementation of program InitSettings
 ********************************************************************)

PROGRAM _INIT

	FOR i := 0 TO 9 BY 1 DO
		DefaultSettingsBU
		(
			BU[i], 	//Bunchunit number
			10, 	//Homespeed
			10,		//MaxPosDev2UseElevator
			50, 	//ReceivePos
			450, 	//ReleasePos
			50, 	//Normal Operation speed
			90, 	//Fast Operation speed
			T#1ms, 	//Drop delay
			T#500ms,//Drop release delay
			0,		//Next chain delay
			92,		//Safe elevator pos start
			246,	//Safe elevator pos start vak
			443,	//Safe elevator pos end vak
			530,	//Safe elevator pos end
			T#500ms	//Bunchbelt pulse
		);

		//Set init _parameters bunchbelts
		BU[i].typBunchBelts.command.iSetSpeed := BU[i].typInterface.iSpeedBunchbelt;
		BU[i].typBunchBelts.command.bEnabledStop := TRUE;
	END_FOR

END_PROGRAM
```

#### Init.var - Local variables
```iecst
(********************************************************************
 * COPYRIGHT -- Microsoft
 ********************************************************************
 * Program: InitSettings
 * File: InitSettingsInit.var
 * Author: jorkes
 * Created: October 27, 2014
 ********************************************************************
 * Local variables of program InitSettings
 ********************************************************************)
VAR
	i : USINT;
END_VAR
```

### Program Logical/BunchUnits/RS_I (IEC) - Reject Station

#### RS_I.st - Implementation code
```iecst
(********************************************************************
 * COPYRIGHT --
 ********************************************************************
 * Program: RS
 * File: RS.st
 * Author: ronspa
 * Created: December 23, 2014
 ********************************************************************
 * Implementation of program RS
 ********************************************************************)

PROGRAM _INIT

(* TODO : Add your code here *)
	RU.usChainPos := SHFTREG.uiRejectPosition;
	RU.typInterface.bEnable := TRUE;
	RU.typSettings.usTimingBU16 := 5; // Pos=7

END_PROGRAM

PROGRAM _CYCLIC

//	IF RU.typInterface.bEnable THEN
//		usGripperIndex := ( SHFTREG.typCounters.usChainCounter + SHFTREG.uiGripperCnt + RU.usChainPos) MOD  SHFTREG.uiGripperCnt;
//		RU.GripperControl.IN := (SHFTREG.typGripper[usGripperIndex].bRejectActive);
//		RU.GripperControl(tiSensDelay := RU.typInterface.tiDelayActiveGripper, tiSensPuls := T#200ms);
//
//		RU.typOUT.bActivateGripper := GripperControl.Q;
//		IF GripperControl.Q THEN
//			IF SHFTREG.typGripper[usGripperIndex].bRejectActive THEN
//				// The reset data must be reset.
//				SHFTREG.typGripper[usGripperIndex].bRejectOnOff := FALSE;
//				SHFTREG.typGripper[usGripperIndex].bRejectActive := FALSE;
//			END_IF
//			RU.typInterface.bEnable := TRUE;
//		END_IF
//	END_IF

END_PROGRAM
```

#### RS_I.var - Local variables
```iecst
(********************************************************************
 * COPYRIGHT --
 ********************************************************************
 * Program: RS
 * File: RS.var
 * Author: ronspa
 * Created: December 23, 2014
 ********************************************************************
 * Local variables of program RS
 ********************************************************************)
VAR
	New_Variable : USINT;
	GripperControl : fbSensControl;
	usGripperIndex : USINT;
END_VAR
```

### Program Logical/BunchUnits/BU_1 (IEC) - Program for Bunch Unit 1

#### BU_1Init.st - Initialization code
```iecst
(********************************************************************
 * COPYRIGHT --
 ********************************************************************
 * Program: BU_1
 * File: BU_1Init.st
 * Author: jorkes
 * Created: September 17, 2014
 ********************************************************************
 * Implementation of program BU_1
 ********************************************************************)

PROGRAM _INIT

	i := 0;

	FOR i := 0 TO 9 DO
		BU[i].typInterface.Status := BU_ST_DISABLED;
		BU[i].usChainPos := SHFTREG.uiBunchUnitPosition[i];

		// For TESTING RSP 23-12-2014

		//Enable 'FI'
		BU[i].typBunchBelts.command.bEnabledStop := TRUE;
		//Bepaal draairichting
		BU[i].typBunchBelts.command.bRunReverse := FALSE;
	END_FOR

	i := 0;
	BU[i].typSettings.usTimingBU16 := 10; // Pos=12
	BU[i].typSettings.usBunchBeltPosition := 0;
END_PROGRAM
```

- BunchUnit.st (reference to Logical/BunchUnits/BU_Ref/BunchUnit.st)

- BunchUnit.var (reference to Logical/BunchUnits/BU_Ref/BunchUnit.var)

### Program Logical/BunchUnits/SC_1 (IEC) - Program for Servo 1

#### SCInit.st - Initialization code
```iecst
(********************************************************************
 * COPYRIGHT --
 ********************************************************************
 * Program: FestoControl
 * File: FestoControlInit.st
 * Author: jorkes
 * Created: September 17, 2014
 ********************************************************************
 * Implementation of program FestoControl
 ********************************************************************)

PROGRAM _INIT

	i := 0;

END_PROGRAM
```

- SC.st (reference to Logical/BunchUnits/SC_Ref/SC.st)

- SC.var (reference to Logical/BunchUnits/SC_Ref/SC.var)

### Program Logical/BunchUnits/BU_2 (IEC) - Program for Bunch Unit 2

#### BU_2Init.st - Initialization code
```iecst
(********************************************************************
 * COPYRIGHT --
 ********************************************************************
 * Program: BU_1
 * File: BU_1Init.st
 * Author: ronspa
 * Created: Januari 12, 2015
 ********************************************************************
 * Implementation of program BU_1
 ********************************************************************)

PROGRAM _INIT

	i := 1;

	BU[i].typInterface.Status := BU_ST_DISABLED;
	BU[i].usChainPos := SHFTREG.uiBunchUnitPosition[i] - 1; // Because position is 0!!!

	// For TESTING RSP 23-12-2014

	//Enable 'FI'
	BU[i].typBunchBelts.command.bEnabledStop := TRUE;
	//Bepaal draairichting
	BU[i].typBunchBelts.command.bRunReverse := FALSE;
	BU[i].typSettings.usTimingBU16 := 14; // Pos=0 ->

END_PROGRAM
```

- BunchUnit.st (reference to Logical/BunchUnits/BU_Ref/BunchUnit.st)

- BunchUnit.var (reference to Logical/BunchUnits/BU_Ref/BunchUnit.var)

### Program Logical/BunchUnits/SC_2 (IEC) - Program for Servo 2

#### SC_2Init.st - Initialization code
```iecst
(********************************************************************
 * COPYRIGHT --
 ********************************************************************
 * Program: SC_2
 * File: SC_2Init.st
 * Author: ronspa
 * Created: February 16, 2015
 ********************************************************************
 * Implementation of program SC_2
 ********************************************************************)

PROGRAM _INIT

	i := 1;

END_PROGRAM
```

- SC.st (reference to Logical/BunchUnits/SC_Ref/SC.st)

- SC.var (reference to Logical/BunchUnits/SC_Ref/SC.var)

### Program Logical/BunchUnits/BU_3 (IEC) - Program for Bunch Unit 3

#### BU_3Init.st - Initialization code
```iecst
(********************************************************************
 * COPYRIGHT --
 ********************************************************************
 * Program: BU_1
 * File: BU_1Init.st
 * Author: ronspa
 * Created: Januari 12, 2015
 ********************************************************************
 * Implementation of program BU_1
 ********************************************************************)

PROGRAM _INIT

	i := 2;

	BU[i].typInterface.Status := BU_ST_DISABLED;
	BU[i].usChainPos := SHFTREG.uiBunchUnitPosition[i] - 1; // Because position is 0!!!

	// For TESTING RSP 23-12-2014

	//Enable 'FI'
	BU[i].typBunchBelts.command.bEnabledStop := TRUE;
	//Bepaal draairichting
	BU[i].typBunchBelts.command.bRunReverse := FALSE;
	BU[i].typSettings.usTimingBU16 := 14; // Pos=0 ->

END_PROGRAM
```

- BunchUnit.st (reference to Logical/BunchUnits/BU_Ref/BunchUnit.st)

- BunchUnit.var (reference to Logical/BunchUnits/BU_Ref/BunchUnit.var)

### Program Logical/BunchUnits/SC_3 (IEC) - Program for Servo 3

#### SC_3Init.st - Initialization code
```iecst
(********************************************************************
 * COPYRIGHT --
 ********************************************************************
 * Program: SC_2
 * File: SC_2Init.st
 * Author: ronspa
 * Created: February 16, 2015
 ********************************************************************
 * Implementation of program SC_2
 ********************************************************************)

PROGRAM _INIT

	i := 2;

END_PROGRAM
```

- SC.st (reference to Logical/BunchUnits/SC_Ref/SC.st)

- SC.var (reference to Logical/BunchUnits/SC_Ref/SC.var)

### Program Logical/BunchUnits/BU_4 (IEC) - Program for Bunch Unit 4

#### BU_4Init.st - Initialization code
```iecst
(********************************************************************
 * COPYRIGHT --
 ********************************************************************
 * Program: BU_1
 * File: BU_1Init.st
 * Author: ronspa
 * Created: Januari 12, 2015
 ********************************************************************
 * Implementation of program BU_1
 ********************************************************************)

PROGRAM _INIT

	i := 3;

	BU[i].typInterface.Status := BU_ST_DISABLED;
	BU[i].usChainPos := SHFTREG.uiBunchUnitPosition[i] - 1; // Because position is 0!!!

	// For TESTING RSP 23-12-2014

	//Enable 'FI'
	BU[i].typBunchBelts.command.bEnabledStop := TRUE;
	//Bepaal draairichting
	BU[i].typBunchBelts.command.bRunReverse := FALSE;
	BU[i].typSettings.usTimingBU16 := 14; // Pos=0 ->

END_PROGRAM
```

- BunchUnit.st (reference to Logical/BunchUnits/BU_Ref/BunchUnit.st)

- BunchUnit.var (reference to Logical/BunchUnits/BU_Ref/BunchUnit.var)

### Program Logical/BunchUnits/SC_4 (IEC) - Program for Servo 4

#### SC_4Init.st - Initialization code
```iecst
(********************************************************************
 * COPYRIGHT --
 ********************************************************************
 * Program: SC_2
 * File: SC_2Init.st
 * Author: ronspa
 * Created: February 16, 2015
 ********************************************************************
 * Implementation of program SC_2
 ********************************************************************)

PROGRAM _INIT

	i := 3;

END_PROGRAM
```

- SC.st (reference to Logical/BunchUnits/SC_Ref/SC.st)

- SC.var (reference to Logical/BunchUnits/SC_Ref/SC.var)

### Program Logical/BunchUnits/BU_5 (IEC) - Program for Bunch Unit 5

#### BU_5Init.st - Initialization code
```iecst
(********************************************************************
 * COPYRIGHT --
 ********************************************************************
 * Program: BU_1
 * File: BU_1Init.st
 * Author: ronspa
 * Created: Januari 12, 2015
 ********************************************************************
 * Implementation of program BU_1
 ********************************************************************)

PROGRAM _INIT

	i := 4;

	BU[i].typInterface.Status := BU_ST_DISABLED;
	BU[i].usChainPos := SHFTREG.uiBunchUnitPosition[i] - 1; // Because position is 0!!!

	// For TESTING RSP 23-12-2014

	//Enable 'FI'
	BU[i].typBunchBelts.command.bEnabledStop := TRUE;
	//Bepaal draairichting
	BU[i].typBunchBelts.command.bRunReverse := FALSE;
	BU[i].typSettings.usTimingBU16 := 14; // Pos=0 ->

END_PROGRAM
```

- BunchUnit.st (reference to Logical/BunchUnits/BU_Ref/BunchUnit.st)

- BunchUnit.var (reference to Logical/BunchUnits/BU_Ref/BunchUnit.var)

### Program Logical/BunchUnits/SC_5 (IEC) - Program for Servo 5

#### SC_5Init.st - Initialization code
```iecst
(********************************************************************
 * COPYRIGHT --
 ********************************************************************
 * Program: SC_2
 * File: SC_2Init.st
 * Author: ronspa
 * Created: February 16, 2015
 ********************************************************************
 * Implementation of program SC_2
 ********************************************************************)

PROGRAM _INIT

	i := 4;

END_PROGRAM
```

- SC.st (reference to Logical/BunchUnits/SC_Ref/SC.st)

- SC.var (reference to Logical/BunchUnits/SC_Ref/SC.var)

### Program Logical/BunchUnits/BU_6 (IEC) - Program for Bunch Unit 6

#### BU_6Init.st - Initialization code
```iecst
(********************************************************************
 * COPYRIGHT --
 ********************************************************************
 * Program: BU_1
 * File: BU_1Init.st
 * Author: ronspa
 * Created: Januari 12, 2015
 ********************************************************************
 * Implementation of program BU_1
 ********************************************************************)

PROGRAM _INIT

	i := 5;

	BU[i].typInterface.Status := BU_ST_DISABLED;
	BU[i].usChainPos := SHFTREG.uiBunchUnitPosition[i] - 1; // Because position is 0!!!

	// For TESTING RSP 23-12-2014

	//Enable 'FI'
	BU[i].typBunchBelts.command.bEnabledStop := TRUE;
	//Bepaal draairichting
	BU[i].typBunchBelts.command.bRunReverse := FALSE;
	BU[i].typSettings.usTimingBU16 := 14; // Pos=0 ->

END_PROGRAM
```

- BunchUnit.st (reference to Logical/BunchUnits/BU_Ref/BunchUnit.st)

- BunchUnit.var (reference to Logical/BunchUnits/BU_Ref/BunchUnit.var)

### Program Logical/BunchUnits/SC_6 (IEC) - Program for Servo 6

#### SC_6Init.st - Initialization code
```iecst
(********************************************************************
 * COPYRIGHT --
 ********************************************************************
 * Program: SC_2
 * File: SC_2Init.st
 * Author: ronspa
 * Created: February 16, 2015
 ********************************************************************
 * Implementation of program SC_2
 ********************************************************************)

PROGRAM _INIT

	i := 5;

END_PROGRAM
```

- SC.st (reference to Logical/BunchUnits/SC_Ref/SC.st)

- SC.var (reference to Logical/BunchUnits/SC_Ref/SC.var)

### Program Logical/BunchUnits/BU_7 (IEC) - Program for Bunch Unit 7

#### BU_7Init.st - Initialization code
```iecst
(********************************************************************
 * COPYRIGHT --
 ********************************************************************
 * Program: BU_1
 * File: BU_1Init.st
 * Author: ronspa
 * Created: Januari 12, 2015
 ********************************************************************
 * Implementation of program BU_1
 ********************************************************************)

PROGRAM _INIT

	i := 6;

	BU[i].typInterface.Status := BU_ST_DISABLED;
	BU[i].usChainPos := SHFTREG.uiBunchUnitPosition[i] - 1; // Because position is 0!!!

	// For TESTING RSP 23-12-2014

	//Enable 'FI'
	BU[i].typBunchBelts.command.bEnabledStop := TRUE;
	//Bepaal draairichting
	BU[i].typBunchBelts.command.bRunReverse := FALSE;
	BU[i].typSettings.usTimingBU16 := 14; // Pos=0 ->

END_PROGRAM
```

- BunchUnit.st (reference to Logical/BunchUnits/BU_Ref/BunchUnit.st)

- BunchUnit.var (reference to Logical/BunchUnits/BU_Ref/BunchUnit.var)

### Program Logical/BunchUnits/SC_7 (IEC) - Program for Servo 7

#### SC_7Init.st - Initialization code
```iecst
(********************************************************************
 * COPYRIGHT --
 ********************************************************************
 * Program: SC_2
 * File: SC_2Init.st
 * Author: ronspa
 * Created: February 16, 2015
 ********************************************************************
 * Implementation of program SC_2
 ********************************************************************)

PROGRAM _INIT

	i := 6;

END_PROGRAM
```

- SC.st (reference to Logical/BunchUnits/SC_Ref/SC.st)

- SC.var (reference to Logical/BunchUnits/SC_Ref/SC.var)

### Program Logical/BunchUnits/BU_8 (IEC) - Program for Bunch Unit 8

#### BU_8Init.st - Initialization code
```iecst
(********************************************************************
 * COPYRIGHT --
 ********************************************************************
 * Program: BU_1
 * File: BU_1Init.st
 * Author: ronspa
 * Created: Januari 12, 2015
 ********************************************************************
 * Implementation of program BU_1
 ********************************************************************)

PROGRAM _INIT

	i := 7;

	BU[i].typInterface.Status := BU_ST_DISABLED;
	BU[i].usChainPos := SHFTREG.uiBunchUnitPosition[i] - 1; // Because position is 0!!!

	// For TESTING RSP 23-12-2014

	//Enable 'FI'
	BU[i].typBunchBelts.command.bEnabledStop := TRUE;
	//Bepaal draairichting
	BU[i].typBunchBelts.command.bRunReverse := FALSE;
	BU[i].typSettings.usTimingBU16 := 14; // Pos=0 ->

END_PROGRAM
```

- BunchUnit.st (reference to Logical/BunchUnits/BU_Ref/BunchUnit.st)

- BunchUnit.var (reference to Logical/BunchUnits/BU_Ref/BunchUnit.var)

### Program Logical/BunchUnits/SC_8 (IEC) - Program for Servo 8

#### SC_8Init.st - Initialization code
```iecst
(********************************************************************
 * COPYRIGHT --
 ********************************************************************
 * Program: SC_2
 * File: SC_2Init.st
 * Author: ronspa
 * Created: February 16, 2015
 ********************************************************************
 * Implementation of program SC_2
 ********************************************************************)

PROGRAM _INIT

	i := 7;

END_PROGRAM
```

- SC.st (reference to Logical/BunchUnits/SC_Ref/SC.st)

- SC.var (reference to Logical/BunchUnits/SC_Ref/SC.var)

### Program Logical/BunchUnits/BU_9 (IEC) - Program for Bunch Unit 3

#### BU_9Init.st - Initialization code
```iecst
(********************************************************************
 * COPYRIGHT --
 ********************************************************************
 * Program: BU_1
 * File: BU_1Init.st
 * Author: ronspa
 * Created: Januari 12, 2015
 ********************************************************************
 * Implementation of program BU_1
 ********************************************************************)

PROGRAM _INIT

	i := 8;

	BU[i].typInterface.Status := BU_ST_DISABLED;
	BU[i].usChainPos := SHFTREG.uiBunchUnitPosition[i] - 1; // Because position is 0!!!

	// For TESTING RSP 23-12-2014

	//Enable 'FI'
	BU[i].typBunchBelts.command.bEnabledStop := TRUE;
	//Bepaal draairichting
	BU[i].typBunchBelts.command.bRunReverse := FALSE;
	BU[i].typSettings.usTimingBU16 := 14; // Pos=0 ->

END_PROGRAM
```

- BunchUnit.st (reference to Logical/BunchUnits/BU_Ref/BunchUnit.st)

- BunchUnit.var (reference to Logical/BunchUnits/BU_Ref/BunchUnit.var)

### Program Logical/BunchUnits/SC_9 (IEC) - Program for Servo 3
